    unicode[3596]:=16#75c8;
    unicode[3597]:=16#75c9;
    unicode[3598]:=16#75ca;
    unicode[3599]:=16#75cd;
    unicode[3600]:=16#75d2;
    unicode[3601]:=16#75d4;
    unicode[3602]:=16#75d5;
    unicode[3603]:=16#75d6;
    unicode[3604]:=16#75d8;
    unicode[3605]:=16#75db;
    unicode[3606]:=16#75de;
    unicode[3607]:=16#75e2;
    unicode[3608]:=16#75e3;
    unicode[3609]:=16#75e4;
    unicode[3610]:=16#75e6;
    unicode[3611]:=16#75e7;
    unicode[3612]:=16#75e8;
    unicode[3613]:=16#75ea;
    unicode[3614]:=16#75eb;
    unicode[3615]:=16#75f0;
    unicode[3616]:=16#75f1;
    unicode[3617]:=16#75f4;
    unicode[3618]:=16#75f9;
    unicode[3619]:=16#75fc;
    unicode[3620]:=16#75ff;
    unicode[3621]:=16#7600;
    unicode[3622]:=16#7601;
    unicode[3623]:=16#7603;
    unicode[3624]:=16#7605;
    unicode[3625]:=16#760a;
    unicode[3626]:=16#760c;
    unicode[3627]:=16#7610;
    unicode[3628]:=16#7615;
    unicode[3629]:=16#7617;
    unicode[3630]:=16#7618;
    unicode[3631]:=16#7619;
    unicode[3632]:=16#761b;
    unicode[3633]:=16#761f;
    unicode[3634]:=16#7620;
    unicode[3635]:=16#7622;
    unicode[3636]:=16#7624;
    unicode[3637]:=16#7625;
    unicode[3638]:=16#7626;
    unicode[3639]:=16#7629;
    unicode[3640]:=16#762a;
    unicode[3641]:=16#762b;
    unicode[3642]:=16#762d;
    unicode[3643]:=16#7630;
    unicode[3644]:=16#7633;
    unicode[3645]:=16#7634;
    unicode[3646]:=16#7635;
    unicode[3647]:=16#7638;
    unicode[3648]:=16#763c;
    unicode[3649]:=16#763e;
    unicode[3650]:=16#763f;
    unicode[3651]:=16#7640;
    unicode[3652]:=16#7643;
    unicode[3653]:=16#764c;
    unicode[3654]:=16#764d;
    unicode[3655]:=16#7654;
    unicode[3656]:=16#7656;
    unicode[3657]:=16#765c;
    unicode[3658]:=16#765e;
    unicode[3659]:=16#7663;
    unicode[3660]:=16#766b;
    unicode[3661]:=16#766f;
    unicode[3662]:=16#7678;
    unicode[3663]:=16#767b;
    unicode[3664]:=16#767d;
    unicode[3665]:=16#767e;
    unicode[3666]:=16#7682;
    unicode[3667]:=16#7684;
    unicode[3668]:=16#7686;
    unicode[3669]:=16#7687;
    unicode[3670]:=16#7688;
    unicode[3671]:=16#768b;
    unicode[3672]:=16#768e;
    unicode[3673]:=16#7691;
    unicode[3674]:=16#7693;
    unicode[3675]:=16#7696;
    unicode[3676]:=16#7699;
    unicode[3677]:=16#76a4;
    unicode[3678]:=16#76ae;
    unicode[3679]:=16#76b1;
    unicode[3680]:=16#76b2;
    unicode[3681]:=16#76b4;
    unicode[3682]:=16#76bf;
    unicode[3683]:=16#76c2;
    unicode[3684]:=16#76c5;
    unicode[3685]:=16#76c6;
    unicode[3686]:=16#76c8;
    unicode[3687]:=16#76ca;
    unicode[3688]:=16#76cd;
    unicode[3689]:=16#76ce;
    unicode[3690]:=16#76cf;
    unicode[3691]:=16#76d0;
    unicode[3692]:=16#76d1;
    unicode[3693]:=16#76d2;
    unicode[3694]:=16#76d4;
    unicode[3695]:=16#76d6;
    unicode[3696]:=16#76d7;
    unicode[3697]:=16#76d8;
    unicode[3698]:=16#76db;
    unicode[3699]:=16#76df;
    unicode[3700]:=16#76e5;
    unicode[3701]:=16#76ee;
    unicode[3702]:=16#76ef;
    unicode[3703]:=16#76f1;
    unicode[3704]:=16#76f2;
    unicode[3705]:=16#76f4;
    unicode[3706]:=16#76f8;
    unicode[3707]:=16#76f9;
    unicode[3708]:=16#76fc;
    unicode[3709]:=16#76fe;
    unicode[3710]:=16#7701;
    unicode[3711]:=16#7704;
    unicode[3712]:=16#7707;
    unicode[3713]:=16#7708;
    unicode[3714]:=16#7709;
    unicode[3715]:=16#770b;
    unicode[3716]:=16#770d;
    unicode[3717]:=16#7719;
    unicode[3718]:=16#771a;
    unicode[3719]:=16#771f;
    unicode[3720]:=16#7720;
    unicode[3721]:=16#7722;
    unicode[3722]:=16#7726;
    unicode[3723]:=16#7728;
    unicode[3724]:=16#7729;
    unicode[3725]:=16#772d;
    unicode[3726]:=16#772f;
    unicode[3727]:=16#7735;
    unicode[3728]:=16#7736;
    unicode[3729]:=16#7737;
    unicode[3730]:=16#7738;
    unicode[3731]:=16#773a;
    unicode[3732]:=16#773c;
    unicode[3733]:=16#7740;
    unicode[3734]:=16#7741;
    unicode[3735]:=16#7743;
    unicode[3736]:=16#7747;
    unicode[3737]:=16#7750;
    unicode[3738]:=16#7751;
    unicode[3739]:=16#775a;
    unicode[3740]:=16#775b;
    unicode[3741]:=16#7761;
    unicode[3742]:=16#7762;
    unicode[3743]:=16#7763;
    unicode[3744]:=16#7765;
    unicode[3745]:=16#7766;
    unicode[3746]:=16#7768;
    unicode[3747]:=16#776b;
    unicode[3748]:=16#776c;
    unicode[3749]:=16#7779;
    unicode[3750]:=16#777d;
    unicode[3751]:=16#777e;
    unicode[3752]:=16#777f;
    unicode[3753]:=16#7780;
    unicode[3754]:=16#7784;
    unicode[3755]:=16#7785;
    unicode[3756]:=16#778c;
    unicode[3757]:=16#778d;
    unicode[3758]:=16#778e;
    unicode[3759]:=16#7791;
    unicode[3760]:=16#7792;
    unicode[3761]:=16#779f;
    unicode[3762]:=16#77a0;
    unicode[3763]:=16#77a2;
    unicode[3764]:=16#77a5;
    unicode[3765]:=16#77a7;
    unicode[3766]:=16#77a9;
    unicode[3767]:=16#77aa;
    unicode[3768]:=16#77ac;
    unicode[3769]:=16#77b0;
    unicode[3770]:=16#77b3;
    unicode[3771]:=16#77b5;
    unicode[3772]:=16#77bb;
    unicode[3773]:=16#77bd;
    unicode[3774]:=16#77bf;
    unicode[3775]:=16#77cd;
    unicode[3776]:=16#77d7;
    unicode[3777]:=16#77db;
    unicode[3778]:=16#77dc;
    unicode[3779]:=16#77e2;
    unicode[3780]:=16#77e3;
    unicode[3781]:=16#77e5;
    unicode[3782]:=16#77e7;
    unicode[3783]:=16#77e9;
    unicode[3784]:=16#77eb;
    unicode[3785]:=16#77ec;
    unicode[3786]:=16#77ed;
    unicode[3787]:=16#77ee;
    unicode[3788]:=16#77f3;
    unicode[3789]:=16#77f6;
    unicode[3790]:=16#77f8;
    unicode[3791]:=16#77fd;
    unicode[3792]:=16#77fe;
    unicode[3793]:=16#77ff;
    unicode[3794]:=16#7800;
    unicode[3795]:=16#7801;
    unicode[3796]:=16#7802;
    unicode[3797]:=16#7809;
    unicode[3798]:=16#780c;
    unicode[3799]:=16#780d;
    unicode[3800]:=16#7811;
    unicode[3801]:=16#7812;
    unicode[3802]:=16#7814;
    unicode[3803]:=16#7816;
    unicode[3804]:=16#7817;
    unicode[3805]:=16#7818;
    unicode[3806]:=16#781a;
    unicode[3807]:=16#781c;
    unicode[3808]:=16#781d;
    unicode[3809]:=16#781f;
    unicode[3810]:=16#7823;
    unicode[3811]:=16#7825;
    unicode[3812]:=16#7826;
    unicode[3813]:=16#7827;
    unicode[3814]:=16#7829;
    unicode[3815]:=16#782c;
    unicode[3816]:=16#782d;
    unicode[3817]:=16#7830;
    unicode[3818]:=16#7834;
    unicode[3819]:=16#7837;
    unicode[3820]:=16#7838;
    unicode[3821]:=16#7839;
    unicode[3822]:=16#783a;
    unicode[3823]:=16#783b;
    unicode[3824]:=16#783c;
    unicode[3825]:=16#783e;
    unicode[3826]:=16#7840;
    unicode[3827]:=16#7845;
    unicode[3828]:=16#7847;
    unicode[3829]:=16#784c;
    unicode[3830]:=16#784e;
    unicode[3831]:=16#7850;
    unicode[3832]:=16#7852;
    unicode[3833]:=16#7855;
    unicode[3834]:=16#7856;
    unicode[3835]:=16#7857;
    unicode[3836]:=16#785d;
    unicode[3837]:=16#786a;
    unicode[3838]:=16#786b;
    unicode[3839]:=16#786c;
    unicode[3840]:=16#786d;
    unicode[3841]:=16#786e;
    unicode[3842]:=16#7877;
    unicode[3843]:=16#787c;
    unicode[3844]:=16#7887;
    unicode[3845]:=16#7889;
    unicode[3846]:=16#788c;
    unicode[3847]:=16#788d;
    unicode[3848]:=16#788e;
    unicode[3849]:=16#7891;
    unicode[3850]:=16#7893;
    unicode[3851]:=16#7897;
    unicode[3852]:=16#7898;
    unicode[3853]:=16#789a;
    unicode[3854]:=16#789b;
    unicode[3855]:=16#789c;
    unicode[3856]:=16#789f;
    unicode[3857]:=16#78a1;
    unicode[3858]:=16#78a3;
    unicode[3859]:=16#78a5;
    unicode[3860]:=16#78a7;
    unicode[3861]:=16#78b0;
    unicode[3862]:=16#78b1;
    unicode[3863]:=16#78b2;
    unicode[3864]:=16#78b3;
    unicode[3865]:=16#78b4;
    unicode[3866]:=16#78b9;
    unicode[3867]:=16#78be;
    unicode[3868]:=16#78c1;
    unicode[3869]:=16#78c5;
    unicode[3870]:=16#78c9;
    unicode[3871]:=16#78ca;
    unicode[3872]:=16#78cb;
    unicode[3873]:=16#78d0;
    unicode[3874]:=16#78d4;
    unicode[3875]:=16#78d5;
    unicode[3876]:=16#78d9;
    unicode[3877]:=16#78e8;
    unicode[3878]:=16#78ec;
    unicode[3879]:=16#78f2;
    unicode[3880]:=16#78f4;
    unicode[3881]:=16#78f7;
    unicode[3882]:=16#78fa;
    unicode[3883]:=16#7901;
    unicode[3884]:=16#7905;
    unicode[3885]:=16#7913;
    unicode[3886]:=16#791e;
    unicode[3887]:=16#7924;
    unicode[3888]:=16#7934;
    unicode[3889]:=16#793a;
    unicode[3890]:=16#793b;
    unicode[3891]:=16#793c;
    unicode[3892]:=16#793e;
    unicode[3893]:=16#7940;
    unicode[3894]:=16#7941;
    unicode[3895]:=16#7946;
    unicode[3896]:=16#7948;
    unicode[3897]:=16#7949;
    unicode[3898]:=16#7953;
    unicode[3899]:=16#7956;
    unicode[3900]:=16#7957;
    unicode[3901]:=16#795a;
    unicode[3902]:=16#795b;
    unicode[3903]:=16#795c;
    unicode[3904]:=16#795d;
    unicode[3905]:=16#795e;
    unicode[3906]:=16#795f;
    unicode[3907]:=16#7960;
    unicode[3908]:=16#7962;
    unicode[3909]:=16#7965;
    unicode[3910]:=16#7967;
    unicode[3911]:=16#7968;
    unicode[3912]:=16#796d;
    unicode[3913]:=16#796f;
    unicode[3914]:=16#7977;
    unicode[3915]:=16#7978;
    unicode[3916]:=16#797a;
    unicode[3917]:=16#7980;
    unicode[3918]:=16#7981;
    unicode[3919]:=16#7984;
    unicode[3920]:=16#7985;
    unicode[3921]:=16#798a;
    unicode[3922]:=16#798f;
    unicode[3923]:=16#799a;
    unicode[3924]:=16#79a7;
    unicode[3925]:=16#79b3;
    unicode[3926]:=16#79b9;
    unicode[3927]:=16#79ba;
    unicode[3928]:=16#79bb;
    unicode[3929]:=16#79bd;
    unicode[3930]:=16#79be;
    unicode[3931]:=16#79c0;
    unicode[3932]:=16#79c1;
    unicode[3933]:=16#79c3;
    unicode[3934]:=16#79c6;
    unicode[3935]:=16#79c9;
    unicode[3936]:=16#79cb;
    unicode[3937]:=16#79cd;
    unicode[3938]:=16#79d1;
    unicode[3939]:=16#79d2;
    unicode[3940]:=16#79d5;
    unicode[3941]:=16#79d8;
    unicode[3942]:=16#79df;
    unicode[3943]:=16#79e3;
    unicode[3944]:=16#79e4;
    unicode[3945]:=16#79e6;
    unicode[3946]:=16#79e7;
    unicode[3947]:=16#79e9;
    unicode[3948]:=16#79eb;
    unicode[3949]:=16#79ed;
    unicode[3950]:=16#79ef;
    unicode[3951]:=16#79f0;
    unicode[3952]:=16#79f8;
    unicode[3953]:=16#79fb;
    unicode[3954]:=16#79fd;
    unicode[3955]:=16#7a00;
    unicode[3956]:=16#7a02;
    unicode[3957]:=16#7a03;
    unicode[3958]:=16#7a06;
    unicode[3959]:=16#7a0b;
    unicode[3960]:=16#7a0d;
    unicode[3961]:=16#7a0e;
    unicode[3962]:=16#7a14;
    unicode[3963]:=16#7a17;
    unicode[3964]:=16#7a1a;
    unicode[3965]:=16#7a1e;
    unicode[3966]:=16#7a20;
    unicode[3967]:=16#7a23;
    unicode[3968]:=16#7a33;
    unicode[3969]:=16#7a37;
    unicode[3970]:=16#7a39;
    unicode[3971]:=16#7a3b;
    unicode[3972]:=16#7a3c;
    unicode[3973]:=16#7a3d;
    unicode[3974]:=16#7a3f;
    unicode[3975]:=16#7a46;
    unicode[3976]:=16#7a51;
    unicode[3977]:=16#7a57;
    unicode[3978]:=16#7a70;
    unicode[3979]:=16#7a74;
    unicode[3980]:=16#7a76;
    unicode[3981]:=16#7a77;
    unicode[3982]:=16#7a78;
    unicode[3983]:=16#7a79;
    unicode[3984]:=16#7a7a;
    unicode[3985]:=16#7a7f;
    unicode[3986]:=16#7a80;
    unicode[3987]:=16#7a81;
    unicode[3988]:=16#7a83;
    unicode[3989]:=16#7a84;
    unicode[3990]:=16#7a86;
    unicode[3991]:=16#7a88;
    unicode[3992]:=16#7a8d;
    unicode[3993]:=16#7a91;
    unicode[3994]:=16#7a92;
    unicode[3995]:=16#7a95;
    unicode[3996]:=16#7a96;
    unicode[3997]:=16#7a97;
    unicode[3998]:=16#7a98;
    unicode[3999]:=16#7a9c;               //unicode码 3000-3999
END_IF;
(* Rung 8 *)
IF P_On THEN
    unicode[4000]:=16#7a9d;
    unicode[4001]:=16#7a9f;
    unicode[4002]:=16#7aa0;
    unicode[4003]:=16#7aa5;
    unicode[4004]:=16#7aa6;
    unicode[4005]:=16#7aa8;
    unicode[4006]:=16#7aac;
    unicode[4007]:=16#7aad;
    unicode[4008]:=16#7ab3;
    unicode[4009]:=16#7abf;
    unicode[4010]:=16#7acb;
    unicode[4011]:=16#7ad6;
    unicode[4012]:=16#7ad9;
    unicode[4013]:=16#7ade;
    unicode[4014]:=16#7adf;
    unicode[4015]:=16#7ae0;
    unicode[4016]:=16#7ae3;
    unicode[4017]:=16#7ae5;
    unicode[4018]:=16#7ae6;
    unicode[4019]:=16#7aed;
    unicode[4020]:=16#7aef;
    unicode[4021]:=16#7af9;
    unicode[4022]:=16#7afa;
    unicode[4023]:=16#7afd;
    unicode[4024]:=16#7aff;
    unicode[4025]:=16#7b03;
    unicode[4026]:=16#7b04;
    unicode[4027]:=16#7b06;
    unicode[4028]:=16#7b08;
    unicode[4029]:=16#7b0a;
    unicode[4030]:=16#7b0b;
    unicode[4031]:=16#7b0f;
    unicode[4032]:=16#7b11;
    unicode[4033]:=16#7b14;
    unicode[4034]:=16#7b15;
    unicode[4035]:=16#7b19;
    unicode[4036]:=16#7b1b;
    unicode[4037]:=16#7b1e;
    unicode[4038]:=16#7b20;
    unicode[4039]:=16#7b24;
    unicode[4040]:=16#7b25;
    unicode[4041]:=16#7b26;
    unicode[4042]:=16#7b28;
    unicode[4043]:=16#7b2a;
    unicode[4044]:=16#7b2b;
    unicode[4045]:=16#7b2c;
    unicode[4046]:=16#7b2e;
    unicode[4047]:=16#7b31;
    unicode[4048]:=16#7b33;
    unicode[4049]:=16#7b38;
    unicode[4050]:=16#7b3a;
    unicode[4051]:=16#7b3c;
    unicode[4052]:=16#7b3e;
    unicode[4053]:=16#7b45;
    unicode[4054]:=16#7b47;
    unicode[4055]:=16#7b49;
    unicode[4056]:=16#7b4b;
    unicode[4057]:=16#7b4c;
    unicode[4058]:=16#7b4f;
    unicode[4059]:=16#7b50;
    unicode[4060]:=16#7b51;
    unicode[4061]:=16#7b52;
    unicode[4062]:=16#7b54;
    unicode[4063]:=16#7b56;
    unicode[4064]:=16#7b58;
    unicode[4065]:=16#7b5a;
    unicode[4066]:=16#7b5b;
    unicode[4067]:=16#7b5d;
    unicode[4068]:=16#7b60;
    unicode[4069]:=16#7b62;
    unicode[4070]:=16#7b6e;
    unicode[4071]:=16#7b71;
    unicode[4072]:=16#7b72;
    unicode[4073]:=16#7b75;
    unicode[4074]:=16#7b77;
    unicode[4075]:=16#7b79;
    unicode[4076]:=16#7b7b;
    unicode[4077]:=16#7b7e;
    unicode[4078]:=16#7b80;
    unicode[4079]:=16#7b85;
    unicode[4080]:=16#7b8d;
    unicode[4081]:=16#7b90;
    unicode[4082]:=16#7b94;
    unicode[4083]:=16#7b95;
    unicode[4084]:=16#7b97;
    unicode[4085]:=16#7b9c;
    unicode[4086]:=16#7b9d;
    unicode[4087]:=16#7ba1;
    unicode[4088]:=16#7ba2;
    unicode[4089]:=16#7ba6;
    unicode[4090]:=16#7ba7;
    unicode[4091]:=16#7ba8;
    unicode[4092]:=16#7ba9;
    unicode[4093]:=16#7baa;
    unicode[4094]:=16#7bab;
    unicode[4095]:=16#7bac;
    unicode[4096]:=16#7bad;
    unicode[4097]:=16#7bb1;
    unicode[4098]:=16#7bb4;
    unicode[4099]:=16#7bb8;
    unicode[4100]:=16#7bc1;
    unicode[4101]:=16#7bc6;
    unicode[4102]:=16#7bc7;
    unicode[4103]:=16#7bcc;
    unicode[4104]:=16#7bd1;
    unicode[4105]:=16#7bd3;
    unicode[4106]:=16#7bd9;
    unicode[4107]:=16#7bda;
    unicode[4108]:=16#7bdd;
    unicode[4109]:=16#7be1;
    unicode[4110]:=16#7be5;
    unicode[4111]:=16#7be6;
    unicode[4112]:=16#7bea;
    unicode[4113]:=16#7bee;
    unicode[4114]:=16#7bf1;
    unicode[4115]:=16#7bf7;
    unicode[4116]:=16#7bfc;
    unicode[4117]:=16#7bfe;
    unicode[4118]:=16#7c07;
    unicode[4119]:=16#7c0b;
    unicode[4120]:=16#7c0c;
    unicode[4121]:=16#7c0f;
    unicode[4122]:=16#7c16;
    unicode[4123]:=16#7c1f;
    unicode[4124]:=16#7c26;
    unicode[4125]:=16#7c27;
    unicode[4126]:=16#7c2a;
    unicode[4127]:=16#7c38;
    unicode[4128]:=16#7c3f;
    unicode[4129]:=16#7c40;
    unicode[4130]:=16#7c41;
    unicode[4131]:=16#7c4d;
    unicode[4132]:=16#7c73;
    unicode[4133]:=16#7c74;
    unicode[4134]:=16#7c7b;
    unicode[4135]:=16#7c7c;
    unicode[4136]:=16#7c7d;
    unicode[4137]:=16#7c89;
    unicode[4138]:=16#7c91;
    unicode[4139]:=16#7c92;
    unicode[4140]:=16#7c95;
    unicode[4141]:=16#7c97;
    unicode[4142]:=16#7c98;
    unicode[4143]:=16#7c9c;
    unicode[4144]:=16#7c9d;
    unicode[4145]:=16#7c9e;
    unicode[4146]:=16#7c9f;
    unicode[4147]:=16#7ca2;
    unicode[4148]:=16#7ca4;
    unicode[4149]:=16#7ca5;
    unicode[4150]:=16#7caa;
    unicode[4151]:=16#7cae;
    unicode[4152]:=16#7cb1;
    unicode[4153]:=16#7cb2;
    unicode[4154]:=16#7cb3;
    unicode[4155]:=16#7cb9;
    unicode[4156]:=16#7cbc;
    unicode[4157]:=16#7cbd;
    unicode[4158]:=16#7cbe;
    unicode[4159]:=16#7cc1;
    unicode[4160]:=16#7cc5;
    unicode[4161]:=16#7cc7;
    unicode[4162]:=16#7cc8;
    unicode[4163]:=16#7cca;
    unicode[4164]:=16#7ccc;
    unicode[4165]:=16#7ccd;
    unicode[4166]:=16#7cd5;
    unicode[4167]:=16#7cd6;
    unicode[4168]:=16#7cd7;
    unicode[4169]:=16#7cd9;
    unicode[4170]:=16#7cdc;
    unicode[4171]:=16#7cdf;
    unicode[4172]:=16#7ce0;
    unicode[4173]:=16#7ce8;
    unicode[4174]:=16#7cef;
    unicode[4175]:=16#7cf8;
    unicode[4176]:=16#7cfb;
    unicode[4177]:=16#7d0a;
    unicode[4178]:=16#7d20;
    unicode[4179]:=16#7d22;
    unicode[4180]:=16#7d27;
    unicode[4181]:=16#7d2b;
    unicode[4182]:=16#7d2f;
    unicode[4183]:=16#7d6e;
    unicode[4184]:=16#7d77;
    unicode[4185]:=16#7da6;
    unicode[4186]:=16#7dae;
    unicode[4187]:=16#7e3b;
    unicode[4188]:=16#7e41;
    unicode[4189]:=16#7e47;
    unicode[4190]:=16#7e82;
    unicode[4191]:=16#7e9b;
    unicode[4192]:=16#7e9f;
    unicode[4193]:=16#7ea0;
    unicode[4194]:=16#7ea1;
    unicode[4195]:=16#7ea2;
    unicode[4196]:=16#7ea3;
    unicode[4197]:=16#7ea4;
    unicode[4198]:=16#7ea5;
    unicode[4199]:=16#7ea6;
    unicode[4200]:=16#7ea7;
    unicode[4201]:=16#7ea8;
    unicode[4202]:=16#7ea9;
    unicode[4203]:=16#7eaa;
    unicode[4204]:=16#7eab;
    unicode[4205]:=16#7eac;
    unicode[4206]:=16#7ead;
    unicode[4207]:=16#7eaf;
    unicode[4208]:=16#7eb0;
    unicode[4209]:=16#7eb1;
    unicode[4210]:=16#7eb2;
    unicode[4211]:=16#7eb3;
    unicode[4212]:=16#7eb5;
    unicode[4213]:=16#7eb6;
    unicode[4214]:=16#7eb7;
    unicode[4215]:=16#7eb8;
    unicode[4216]:=16#7eb9;
    unicode[4217]:=16#7eba;
    unicode[4218]:=16#7ebd;
    unicode[4219]:=16#7ebe;
    unicode[4220]:=16#7ebf;
    unicode[4221]:=16#7ec0;
    unicode[4222]:=16#7ec1;
    unicode[4223]:=16#7ec2;
    unicode[4224]:=16#7ec3;
    unicode[4225]:=16#7ec4;
    unicode[4226]:=16#7ec5;
    unicode[4227]:=16#7ec6;
    unicode[4228]:=16#7ec7;
    unicode[4229]:=16#7ec8;
    unicode[4230]:=16#7ec9;
    unicode[4231]:=16#7eca;
    unicode[4232]:=16#7ecb;
    unicode[4233]:=16#7ecc;
    unicode[4234]:=16#7ecd;
    unicode[4235]:=16#7ece;
    unicode[4236]:=16#7ecf;
    unicode[4237]:=16#7ed0;
    unicode[4238]:=16#7ed1;
    unicode[4239]:=16#7ed2;
    unicode[4240]:=16#7ed3;
    unicode[4241]:=16#7ed4;
    unicode[4242]:=16#7ed5;
    unicode[4243]:=16#7ed7;
    unicode[4244]:=16#7ed8;
    unicode[4245]:=16#7ed9;
    unicode[4246]:=16#7eda;
    unicode[4247]:=16#7edb;
    unicode[4248]:=16#7edc;
    unicode[4249]:=16#7edd;
    unicode[4250]:=16#7ede;
    unicode[4251]:=16#7edf;
    unicode[4252]:=16#7ee0;
    unicode[4253]:=16#7ee1;
    unicode[4254]:=16#7ee2;
    unicode[4255]:=16#7ee3;
    unicode[4256]:=16#7ee5;
    unicode[4257]:=16#7ee6;
    unicode[4258]:=16#7ee7;
    unicode[4259]:=16#7ee8;
    unicode[4260]:=16#7ee9;
    unicode[4261]:=16#7eea;
    unicode[4262]:=16#7eeb;
    unicode[4263]:=16#7eed;
    unicode[4264]:=16#7eee;
    unicode[4265]:=16#7eef;
    unicode[4266]:=16#7ef0;
    unicode[4267]:=16#7ef1;
    unicode[4268]:=16#7ef2;
    unicode[4269]:=16#7ef3;
    unicode[4270]:=16#7ef4;
    unicode[4271]:=16#7ef5;
    unicode[4272]:=16#7ef6;
    unicode[4273]:=16#7ef7;
    unicode[4274]:=16#7ef8;
    unicode[4275]:=16#7efa;
    unicode[4276]:=16#7efb;
    unicode[4277]:=16#7efc;
    unicode[4278]:=16#7efd;
    unicode[4279]:=16#7efe;
    unicode[4280]:=16#7eff;
    unicode[4281]:=16#7f00;
    unicode[4282]:=16#7f01;
    unicode[4283]:=16#7f02;
    unicode[4284]:=16#7f03;
    unicode[4285]:=16#7f04;
    unicode[4286]:=16#7f05;
    unicode[4287]:=16#7f06;
    unicode[4288]:=16#7f07;
    unicode[4289]:=16#7f08;
    unicode[4290]:=16#7f09;
    unicode[4291]:=16#7f0b;
    unicode[4292]:=16#7f0c;
    unicode[4293]:=16#7f0d;
    unicode[4294]:=16#7f0e;
    unicode[4295]:=16#7f0f;
    unicode[4296]:=16#7f11;
    unicode[4297]:=16#7f12;
    unicode[4298]:=16#7f13;
    unicode[4299]:=16#7f14;
    unicode[4300]:=16#7f15;
    unicode[4301]:=16#7f16;
    unicode[4302]:=16#7f17;
    unicode[4303]:=16#7f18;
    unicode[4304]:=16#7f19;
    unicode[4305]:=16#7f1a;
    unicode[4306]:=16#7f1b;
    unicode[4307]:=16#7f1c;
    unicode[4308]:=16#7f1d;
    unicode[4309]:=16#7f1f;
    unicode[4310]:=16#7f20;
    unicode[4311]:=16#7f21;
    unicode[4312]:=16#7f22;
    unicode[4313]:=16#7f23;
    unicode[4314]:=16#7f24;
    unicode[4315]:=16#7f25;
    unicode[4316]:=16#7f26;
    unicode[4317]:=16#7f27;
    unicode[4318]:=16#7f28;
    unicode[4319]:=16#7f29;
    unicode[4320]:=16#7f2a;
    unicode[4321]:=16#7f2b;
    unicode[4322]:=16#7f2c;
    unicode[4323]:=16#7f2d;
    unicode[4324]:=16#7f2e;
    unicode[4325]:=16#7f2f;
    unicode[4326]:=16#7f30;
    unicode[4327]:=16#7f31;
    unicode[4328]:=16#7f32;
    unicode[4329]:=16#7f33;
    unicode[4330]:=16#7f34;
    unicode[4331]:=16#7f35;
    unicode[4332]:=16#7f36;
    unicode[4333]:=16#7f38;
    unicode[4334]:=16#7f3a;
    unicode[4335]:=16#7f42;
    unicode[4336]:=16#7f44;
    unicode[4337]:=16#7f45;
    unicode[4338]:=16#7f50;
    unicode[4339]:=16#7f51;
    unicode[4340]:=16#7f54;
    unicode[4341]:=16#7f55;
    unicode[4342]:=16#7f57;
    unicode[4343]:=16#7f58;
    unicode[4344]:=16#7f5a;
    unicode[4345]:=16#7f5f;
    unicode[4346]:=16#7f61;
    unicode[4347]:=16#7f62;
    unicode[4348]:=16#7f68;
    unicode[4349]:=16#7f69;
    unicode[4350]:=16#7f6a;
    unicode[4351]:=16#7f6e;
    unicode[4352]:=16#7f71;
    unicode[4353]:=16#7f72;
    unicode[4354]:=16#7f74;
    unicode[4355]:=16#7f79;
    unicode[4356]:=16#7f7e;
    unicode[4357]:=16#7f81;
    unicode[4358]:=16#7f8a;
    unicode[4359]:=16#7f8c;
    unicode[4360]:=16#7f8e;
    unicode[4361]:=16#7f94;
    unicode[4362]:=16#7f9a;
    unicode[4363]:=16#7f9d;
    unicode[4364]:=16#7f9e;
    unicode[4365]:=16#7f9f;
    unicode[4366]:=16#7fa1;
    unicode[4367]:=16#7fa4;
    unicode[4368]:=16#7fa7;
    unicode[4369]:=16#7faf;
    unicode[4370]:=16#7fb0;
    unicode[4371]:=16#7fb2;
    unicode[4372]:=16#7fb8;
    unicode[4373]:=16#7fb9;
    unicode[4374]:=16#7fbc;
    unicode[4375]:=16#7fbd;
    unicode[4376]:=16#7fbf;
    unicode[4377]:=16#7fc1;
    unicode[4378]:=16#7fc5;
    unicode[4379]:=16#7fca;
    unicode[4380]:=16#7fcc;
    unicode[4381]:=16#7fce;
    unicode[4382]:=16#7fd4;
    unicode[4383]:=16#7fd5;
    unicode[4384]:=16#7fd8;
    unicode[4385]:=16#7fdf;
    unicode[4386]:=16#7fe0;
    unicode[4387]:=16#7fe1;
    unicode[4388]:=16#7fe5;
    unicode[4389]:=16#7fe6;
    unicode[4390]:=16#7fe9;
    unicode[4391]:=16#7fee;
    unicode[4392]:=16#7ff0;
    unicode[4393]:=16#7ff1;
    unicode[4394]:=16#7ff3;
    unicode[4395]:=16#7ffb;
    unicode[4396]:=16#7ffc;
    unicode[4397]:=16#8000;
    unicode[4398]:=16#8001;
    unicode[4399]:=16#8003;
    unicode[4400]:=16#8004;
    unicode[4401]:=16#8005;
    unicode[4402]:=16#8006;
    unicode[4403]:=16#800b;
    unicode[4404]:=16#800c;
    unicode[4405]:=16#800d;
    unicode[4406]:=16#8010;
    unicode[4407]:=16#8012;
    unicode[4408]:=16#8014;
    unicode[4409]:=16#8015;
    unicode[4410]:=16#8016;
    unicode[4411]:=16#8017;
    unicode[4412]:=16#8018;
    unicode[4413]:=16#8019;
    unicode[4414]:=16#801c;
    unicode[4415]:=16#8020;
    unicode[4416]:=16#8022;
    unicode[4417]:=16#8025;
    unicode[4418]:=16#8026;
    unicode[4419]:=16#8027;
    unicode[4420]:=16#8028;
    unicode[4421]:=16#8029;
    unicode[4422]:=16#802a;
    unicode[4423]:=16#8031;
    unicode[4424]:=16#8033;
    unicode[4425]:=16#8035;
    unicode[4426]:=16#8036;
    unicode[4427]:=16#8037;
    unicode[4428]:=16#8038;
    unicode[4429]:=16#803b;
    unicode[4430]:=16#803d;
    unicode[4431]:=16#803f;
    unicode[4432]:=16#8042;
    unicode[4433]:=16#8043;
    unicode[4434]:=16#8046;
    unicode[4435]:=16#804a;
    unicode[4436]:=16#804b;
    unicode[4437]:=16#804c;
    unicode[4438]:=16#804d;
    unicode[4439]:=16#8052;
    unicode[4440]:=16#8054;
    unicode[4441]:=16#8058;
    unicode[4442]:=16#805a;
    unicode[4443]:=16#8069;
    unicode[4444]:=16#806a;
    unicode[4445]:=16#8071;
    unicode[4446]:=16#807f;
    unicode[4447]:=16#8080;
    unicode[4448]:=16#8083;
    unicode[4449]:=16#8084;
    unicode[4450]:=16#8086;
    unicode[4451]:=16#8087;
    unicode[4452]:=16#8089;
    unicode[4453]:=16#808b;
    unicode[4454]:=16#808c;
    unicode[4455]:=16#8093;
    unicode[4456]:=16#8096;
    unicode[4457]:=16#8098;
    unicode[4458]:=16#809a;
    unicode[4459]:=16#809b;
    unicode[4460]:=16#809c;
    unicode[4461]:=16#809d;
    unicode[4462]:=16#809f;
    unicode[4463]:=16#80a0;
    unicode[4464]:=16#80a1;
    unicode[4465]:=16#80a2;
    unicode[4466]:=16#80a4;
    unicode[4467]:=16#80a5;
    unicode[4468]:=16#80a9;
    unicode[4469]:=16#80aa;
    unicode[4470]:=16#80ab;
    unicode[4471]:=16#80ad;
    unicode[4472]:=16#80ae;
    unicode[4473]:=16#80af;
    unicode[4474]:=16#80b1;
    unicode[4475]:=16#80b2;
    unicode[4476]:=16#80b4;
    unicode[4477]:=16#80b7;
    unicode[4478]:=16#80ba;
    unicode[4479]:=16#80bc;
    unicode[4480]:=16#80bd;
    unicode[4481]:=16#80be;
    unicode[4482]:=16#80bf;
    unicode[4483]:=16#80c0;
    unicode[4484]:=16#80c1;
    unicode[4485]:=16#80c2;
    unicode[4486]:=16#80c3;
    unicode[4487]:=16#80c4;
    unicode[4488]:=16#80c6;
    unicode[4489]:=16#80cc;
    unicode[4490]:=16#80cd;
    unicode[4491]:=16#80ce;
    unicode[4492]:=16#80d6;
    unicode[4493]:=16#80d7;
    unicode[4494]:=16#80d9;
    unicode[4495]:=16#80da;
    unicode[4496]:=16#80db;
    unicode[4497]:=16#80dc;
    unicode[4498]:=16#80dd;
    unicode[4499]:=16#80de;
    unicode[4500]:=16#80e1;
    unicode[4501]:=16#80e4;
    unicode[4502]:=16#80e5;
    unicode[4503]:=16#80e7;
    unicode[4504]:=16#80e8;
    unicode[4505]:=16#80e9;
    unicode[4506]:=16#80ea;
    unicode[4507]:=16#80eb;
    unicode[4508]:=16#80ec;
    unicode[4509]:=16#80ed;
    unicode[4510]:=16#80ef;
    unicode[4511]:=16#80f0;
    unicode[4512]:=16#80f1;
    unicode[4513]:=16#80f2;
    unicode[4514]:=16#80f3;
    unicode[4515]:=16#80f4;
    unicode[4516]:=16#80f6;
    unicode[4517]:=16#80f8;
    unicode[4518]:=16#80fa;
    unicode[4519]:=16#80fc;
    unicode[4520]:=16#80fd;
    unicode[4521]:=16#8102;
    unicode[4522]:=16#8106;
    unicode[4523]:=16#8109;
    unicode[4524]:=16#810a;
    unicode[4525]:=16#810d;
    unicode[4526]:=16#810e;
    unicode[4527]:=16#810f;
    unicode[4528]:=16#8110;
    unicode[4529]:=16#8111;
    unicode[4530]:=16#8112;
    unicode[4531]:=16#8113;
    unicode[4532]:=16#8114;
    unicode[4533]:=16#8116;
    unicode[4534]:=16#8118;
    unicode[4535]:=16#811a;
    unicode[4536]:=16#811e;
    unicode[4537]:=16#812c;
    unicode[4538]:=16#812f;
    unicode[4539]:=16#8131;
    unicode[4540]:=16#8132;
    unicode[4541]:=16#8136;
    unicode[4542]:=16#8138;
    unicode[4543]:=16#813e;
    unicode[4544]:=16#8146;
    unicode[4545]:=16#8148;
    unicode[4546]:=16#814a;
    unicode[4547]:=16#814b;
    unicode[4548]:=16#814c;
    unicode[4549]:=16#8150;
    unicode[4550]:=16#8151;
    unicode[4551]:=16#8153;
    unicode[4552]:=16#8154;
    unicode[4553]:=16#8155;
    unicode[4554]:=16#8159;
    unicode[4555]:=16#815a;
    unicode[4556]:=16#8160;
    unicode[4557]:=16#8165;
    unicode[4558]:=16#8167;
    unicode[4559]:=16#8169;
    unicode[4560]:=16#816d;
    unicode[4561]:=16#816e;
    unicode[4562]:=16#8170;
    unicode[4563]:=16#8171;
    unicode[4564]:=16#8174;
    unicode[4565]:=16#8179;
    unicode[4566]:=16#817a;
    unicode[4567]:=16#817b;
    unicode[4568]:=16#817c;
    unicode[4569]:=16#817d;
    unicode[4570]:=16#817e;
    unicode[4571]:=16#817f;
    unicode[4572]:=16#8180;
    unicode[4573]:=16#8182;
    unicode[4574]:=16#8188;
    unicode[4575]:=16#818a;
    unicode[4576]:=16#818f;
    unicode[4577]:=16#8191;
    unicode[4578]:=16#8198;
    unicode[4579]:=16#819b;
    unicode[4580]:=16#819c;
    unicode[4581]:=16#819d;
    unicode[4582]:=16#81a3;
    unicode[4583]:=16#81a6;
    unicode[4584]:=16#81a8;
    unicode[4585]:=16#81aa;
    unicode[4586]:=16#81b3;
    unicode[4587]:=16#81ba;
    unicode[4588]:=16#81bb;
    unicode[4589]:=16#81c0;
    unicode[4590]:=16#81c1;
    unicode[4591]:=16#81c2;
    unicode[4592]:=16#81c3;
    unicode[4593]:=16#81c6;
    unicode[4594]:=16#81ca;
    unicode[4595]:=16#81cc;
    unicode[4596]:=16#81e3;
    unicode[4597]:=16#81e7;
    unicode[4598]:=16#81ea;
    unicode[4599]:=16#81ec;
    unicode[4600]:=16#81ed;
    unicode[4601]:=16#81f3;
    unicode[4602]:=16#81f4;
    unicode[4603]:=16#81fb;
    unicode[4604]:=16#81fc;
    unicode[4605]:=16#81fe;
    unicode[4606]:=16#8200;
    unicode[4607]:=16#8201;
    unicode[4608]:=16#8202;
    unicode[4609]:=16#8204;
    unicode[4610]:=16#8205;
    unicode[4611]:=16#8206;
    unicode[4612]:=16#820c;
    unicode[4613]:=16#820d;
    unicode[4614]:=16#8210;
    unicode[4615]:=16#8212;
    unicode[4616]:=16#8214;
    unicode[4617]:=16#821b;
    unicode[4618]:=16#821c;
    unicode[4619]:=16#821e;
    unicode[4620]:=16#821f;
    unicode[4621]:=16#8221;
    unicode[4622]:=16#8222;
    unicode[4623]:=16#8223;
    unicode[4624]:=16#8228;
    unicode[4625]:=16#822a;
    unicode[4626]:=16#822b;
    unicode[4627]:=16#822c;
    unicode[4628]:=16#822d;
    unicode[4629]:=16#822f;
    unicode[4630]:=16#8230;
    unicode[4631]:=16#8231;
    unicode[4632]:=16#8233;
    unicode[4633]:=16#8234;
    unicode[4634]:=16#8235;
    unicode[4635]:=16#8236;
    unicode[4636]:=16#8237;
    unicode[4637]:=16#8238;
    unicode[4638]:=16#8239;
    unicode[4639]:=16#823b;
    unicode[4640]:=16#823e;
    unicode[4641]:=16#8244;
    unicode[4642]:=16#8247;
    unicode[4643]:=16#8249;
    unicode[4644]:=16#824b;
    unicode[4645]:=16#824f;
    unicode[4646]:=16#8258;
    unicode[4647]:=16#825a;
    unicode[4648]:=16#825f;
    unicode[4649]:=16#8268;
    unicode[4650]:=16#826e;
    unicode[4651]:=16#826f;
    unicode[4652]:=16#8270;
    unicode[4653]:=16#8272;
    unicode[4654]:=16#8273;
    unicode[4655]:=16#8274;
    unicode[4656]:=16#8279;
    unicode[4657]:=16#827a;
    unicode[4658]:=16#827d;
    unicode[4659]:=16#827e;
    unicode[4660]:=16#827f;
    unicode[4661]:=16#8282;
    unicode[4662]:=16#8284;
    unicode[4663]:=16#8288;
    unicode[4664]:=16#828a;
    unicode[4665]:=16#828b;
    unicode[4666]:=16#828d;
    unicode[4667]:=16#828e;
    unicode[4668]:=16#828f;
    unicode[4669]:=16#8291;
    unicode[4670]:=16#8292;
    unicode[4671]:=16#8297;
    unicode[4672]:=16#8298;
    unicode[4673]:=16#8299;
    unicode[4674]:=16#829c;
    unicode[4675]:=16#829d;
    unicode[4676]:=16#829f;
    unicode[4677]:=16#82a1;
    unicode[4678]:=16#82a4;
    unicode[4679]:=16#82a5;
    unicode[4680]:=16#82a6;
    unicode[4681]:=16#82a8;
    unicode[4682]:=16#82a9;
    unicode[4683]:=16#82aa;
    unicode[4684]:=16#82ab;
    unicode[4685]:=16#82ac;
    unicode[4686]:=16#82ad;
    unicode[4687]:=16#82ae;
    unicode[4688]:=16#82af;
    unicode[4689]:=16#82b0;
    unicode[4690]:=16#82b1;
    unicode[4691]:=16#82b3;
    unicode[4692]:=16#82b4;
    unicode[4693]:=16#82b7;
    unicode[4694]:=16#82b8;
    unicode[4695]:=16#82b9;
    unicode[4696]:=16#82bd;
    unicode[4697]:=16#82be;
    unicode[4698]:=16#82c1;
    unicode[4699]:=16#82c4;
    unicode[4700]:=16#82c7;
    unicode[4701]:=16#82c8;
    unicode[4702]:=16#82ca;
    unicode[4703]:=16#82cb;
    unicode[4704]:=16#82cc;
    unicode[4705]:=16#82cd;
    unicode[4706]:=16#82ce;
    unicode[4707]:=16#82cf;
    unicode[4708]:=16#82d1;
    unicode[4709]:=16#82d2;
    unicode[4710]:=16#82d3;
    unicode[4711]:=16#82d4;
    unicode[4712]:=16#82d5;
    unicode[4713]:=16#82d7;
    unicode[4714]:=16#82d8;
    unicode[4715]:=16#82db;
    unicode[4716]:=16#82dc;
    unicode[4717]:=16#82de;
    unicode[4718]:=16#82df;
    unicode[4719]:=16#82e0;
    unicode[4720]:=16#82e1;
    unicode[4721]:=16#82e3;
    unicode[4722]:=16#82e4;
    unicode[4723]:=16#82e5;
    unicode[4724]:=16#82e6;
    unicode[4725]:=16#82eb;
    unicode[4726]:=16#82ef;
    unicode[4727]:=16#82f1;
    unicode[4728]:=16#82f4;
    unicode[4729]:=16#82f7;
    unicode[4730]:=16#82f9;
    unicode[4731]:=16#82fb;
    unicode[4732]:=16#8301;
    unicode[4733]:=16#8302;
    unicode[4734]:=16#8303;
    unicode[4735]:=16#8304;
    unicode[4736]:=16#8305;
    unicode[4737]:=16#8306;
    unicode[4738]:=16#8307;
    unicode[4739]:=16#8308;
    unicode[4740]:=16#8309;
    unicode[4741]:=16#830c;
    unicode[4742]:=16#830e;
    unicode[4743]:=16#830f;
    unicode[4744]:=16#8311;
    unicode[4745]:=16#8314;
    unicode[4746]:=16#8315;
    unicode[4747]:=16#8317;
    unicode[4748]:=16#831a;
    unicode[4749]:=16#831b;
    unicode[4750]:=16#831c;
    unicode[4751]:=16#8327;
    unicode[4752]:=16#8328;
    unicode[4753]:=16#832b;
    unicode[4754]:=16#832c;
    unicode[4755]:=16#832d;
    unicode[4756]:=16#832f;
    unicode[4757]:=16#8331;
    unicode[4758]:=16#8333;
    unicode[4759]:=16#8334;
    unicode[4760]:=16#8335;
    unicode[4761]:=16#8336;
    unicode[4762]:=16#8338;
    unicode[4763]:=16#8339;
    unicode[4764]:=16#833a;
    unicode[4765]:=16#833c;
    unicode[4766]:=16#8340;
    unicode[4767]:=16#8343;
    unicode[4768]:=16#8346;
    unicode[4769]:=16#8347;
    unicode[4770]:=16#8349;
    unicode[4771]:=16#834f;
    unicode[4772]:=16#8350;
    unicode[4773]:=16#8351;
    unicode[4774]:=16#8352;
    unicode[4775]:=16#8354;
    unicode[4776]:=16#835a;
    unicode[4777]:=16#835b;
    unicode[4778]:=16#835c;
    unicode[4779]:=16#835e;
    unicode[4780]:=16#835f;
    unicode[4781]:=16#8360;
    unicode[4782]:=16#8361;
    unicode[4783]:=16#8363;
    unicode[4784]:=16#8364;
    unicode[4785]:=16#8365;
    unicode[4786]:=16#8366;
    unicode[4787]:=16#8367;
    unicode[4788]:=16#8368;
    unicode[4789]:=16#8369;
    unicode[4790]:=16#836a;
    unicode[4791]:=16#836b;
    unicode[4792]:=16#836c;
    unicode[4793]:=16#836d;
    unicode[4794]:=16#836e;
    unicode[4795]:=16#836f;
    unicode[4796]:=16#8377;
    unicode[4797]:=16#8378;
    unicode[4798]:=16#837b;
    unicode[4799]:=16#837c;
    unicode[4800]:=16#837d;
    unicode[4801]:=16#8385;
    unicode[4802]:=16#8386;
    unicode[4803]:=16#8389;
    unicode[4804]:=16#838e;
    unicode[4805]:=16#8392;
    unicode[4806]:=16#8393;
    unicode[4807]:=16#8398;
    unicode[4808]:=16#839b;
    unicode[4809]:=16#839c;
    unicode[4810]:=16#839e;
    unicode[4811]:=16#83a0;
    unicode[4812]:=16#83a8;
    unicode[4813]:=16#83a9;
    unicode[4814]:=16#83aa;
    unicode[4815]:=16#83ab;
    unicode[4816]:=16#83b0;
    unicode[4817]:=16#83b1;
    unicode[4818]:=16#83b2;
    unicode[4819]:=16#83b3;
    unicode[4820]:=16#83b4;
    unicode[4821]:=16#83b6;
    unicode[4822]:=16#83b7;
    unicode[4823]:=16#83b8;
    unicode[4824]:=16#83b9;
    unicode[4825]:=16#83ba;
    unicode[4826]:=16#83bc;
    unicode[4827]:=16#83bd;
    unicode[4828]:=16#83c0;
    unicode[4829]:=16#83c1;
    unicode[4830]:=16#83c5;
    unicode[4831]:=16#83c7;
    unicode[4832]:=16#83ca;
    unicode[4833]:=16#83cc;
    unicode[4834]:=16#83cf;
    unicode[4835]:=16#83d4;
    unicode[4836]:=16#83d6;
    unicode[4837]:=16#83d8;
    unicode[4838]:=16#83dc;
    unicode[4839]:=16#83dd;
    unicode[4840]:=16#83df;
    unicode[4841]:=16#83e0;
    unicode[4842]:=16#83e1;
    unicode[4843]:=16#83e5;
    unicode[4844]:=16#83e9;
    unicode[4845]:=16#83ea;
    unicode[4846]:=16#83f0;
    unicode[4847]:=16#83f1;
    unicode[4848]:=16#83f2;
    unicode[4849]:=16#83f8;
    unicode[4850]:=16#83f9;
    unicode[4851]:=16#83fd;
    unicode[4852]:=16#8401;
    unicode[4853]:=16#8403;
    unicode[4854]:=16#8404;
    unicode[4855]:=16#8406;
    unicode[4856]:=16#840b;
    unicode[4857]:=16#840c;
    unicode[4858]:=16#840d;
    unicode[4859]:=16#840e;
    unicode[4860]:=16#840f;
    unicode[4861]:=16#8411;
    unicode[4862]:=16#8418;
    unicode[4863]:=16#841c;
    unicode[4864]:=16#841d;
    unicode[4865]:=16#8424;
    unicode[4866]:=16#8425;
    unicode[4867]:=16#8426;
    unicode[4868]:=16#8427;
    unicode[4869]:=16#8428;
    unicode[4870]:=16#8431;
    unicode[4871]:=16#8438;
    unicode[4872]:=16#843c;
    unicode[4873]:=16#843d;
    unicode[4874]:=16#8446;
    unicode[4875]:=16#8451;
    unicode[4876]:=16#8457;
    unicode[4877]:=16#8459;
    unicode[4878]:=16#845a;
    unicode[4879]:=16#845b;
    unicode[4880]:=16#845c;
    unicode[4881]:=16#8461;
    unicode[4882]:=16#8463;
    unicode[4883]:=16#8469;
    unicode[4884]:=16#846b;
    unicode[4885]:=16#846c;
    unicode[4886]:=16#846d;
    unicode[4887]:=16#8471;
    unicode[4888]:=16#8473;
    unicode[4889]:=16#8475;
    unicode[4890]:=16#8476;
    unicode[4891]:=16#8478;
    unicode[4892]:=16#847a;
    unicode[4893]:=16#8482;
    unicode[4894]:=16#8487;
    unicode[4895]:=16#8488;
    unicode[4896]:=16#8489;
    unicode[4897]:=16#848b;
    unicode[4898]:=16#848c;
    unicode[4899]:=16#848e;
    unicode[4900]:=16#8497;
    unicode[4901]:=16#8499;
    unicode[4902]:=16#849c;
    unicode[4903]:=16#84a1;
    unicode[4904]:=16#84af;
    unicode[4905]:=16#84b2;
    unicode[4906]:=16#84b4;
    unicode[4907]:=16#84b8;
    unicode[4908]:=16#84b9;
    unicode[4909]:=16#84ba;
    unicode[4910]:=16#84bd;
    unicode[4911]:=16#84bf;
    unicode[4912]:=16#84c1;
    unicode[4913]:=16#84c4;
    unicode[4914]:=16#84c9;
    unicode[4915]:=16#84ca;
    unicode[4916]:=16#84cd;
    unicode[4917]:=16#84d0;
    unicode[4918]:=16#84d1;
    unicode[4919]:=16#84d3;
    unicode[4920]:=16#84d6;
    unicode[4921]:=16#84dd;
    unicode[4922]:=16#84df;
    unicode[4923]:=16#84e0;
    unicode[4924]:=16#84e3;
    unicode[4925]:=16#84e5;
    unicode[4926]:=16#84e6;
    unicode[4927]:=16#84ec;
    unicode[4928]:=16#84f0;
    unicode[4929]:=16#84fc;
    unicode[4930]:=16#84ff;
    unicode[4931]:=16#850c;
    unicode[4932]:=16#8511;
    unicode[4933]:=16#8513;
    unicode[4934]:=16#8517;
    unicode[4935]:=16#851a;
    unicode[4936]:=16#851f;
    unicode[4937]:=16#8521;
    unicode[4938]:=16#852b;
    unicode[4939]:=16#852c;
    unicode[4940]:=16#8537;
    unicode[4941]:=16#8538;
    unicode[4942]:=16#8539;
    unicode[4943]:=16#853a;
    unicode[4944]:=16#853b;
    unicode[4945]:=16#853c;
    unicode[4946]:=16#853d;
    unicode[4947]:=16#8543;
    unicode[4948]:=16#8548;
    unicode[4949]:=16#8549;
    unicode[4950]:=16#854a;
    unicode[4951]:=16#8556;
    unicode[4952]:=16#8559;
    unicode[4953]:=16#855e;
    unicode[4954]:=16#8564;
    unicode[4955]:=16#8568;
    unicode[4956]:=16#8572;
    unicode[4957]:=16#8574;
    unicode[4958]:=16#8579;
    unicode[4959]:=16#857a;
    unicode[4960]:=16#857b;
    unicode[4961]:=16#857e;
    unicode[4962]:=16#8584;
    unicode[4963]:=16#8585;
    unicode[4964]:=16#8587;
    unicode[4965]:=16#858f;
    unicode[4966]:=16#859b;
    unicode[4967]:=16#859c;
    unicode[4968]:=16#85a4;
    unicode[4969]:=16#85a8;
    unicode[4970]:=16#85aa;
    unicode[4971]:=16#85ae;
    unicode[4972]:=16#85af;
    unicode[4973]:=16#85b0;
    unicode[4974]:=16#85b7;
    unicode[4975]:=16#85b9;
    unicode[4976]:=16#85c1;
    unicode[4977]:=16#85c9;
    unicode[4978]:=16#85cf;
    unicode[4979]:=16#85d0;
    unicode[4980]:=16#85d3;
    unicode[4981]:=16#85d5;
    unicode[4982]:=16#85dc;
    unicode[4983]:=16#85e4;
    unicode[4984]:=16#85e9;
    unicode[4985]:=16#85fb;
    unicode[4986]:=16#85ff;
    unicode[4987]:=16#8605;
    unicode[4988]:=16#8611;
    unicode[4989]:=16#8616;
    unicode[4990]:=16#8627;
    unicode[4991]:=16#8629;
    unicode[4992]:=16#8638;
    unicode[4993]:=16#863c;
    unicode[4994]:=16#864d;
    unicode[4995]:=16#864e;
    unicode[4996]:=16#864f;
    unicode[4997]:=16#8650;
    unicode[4998]:=16#8651;
    unicode[4999]:=16#8654;           //unicode码 4000-4999
END_IF;

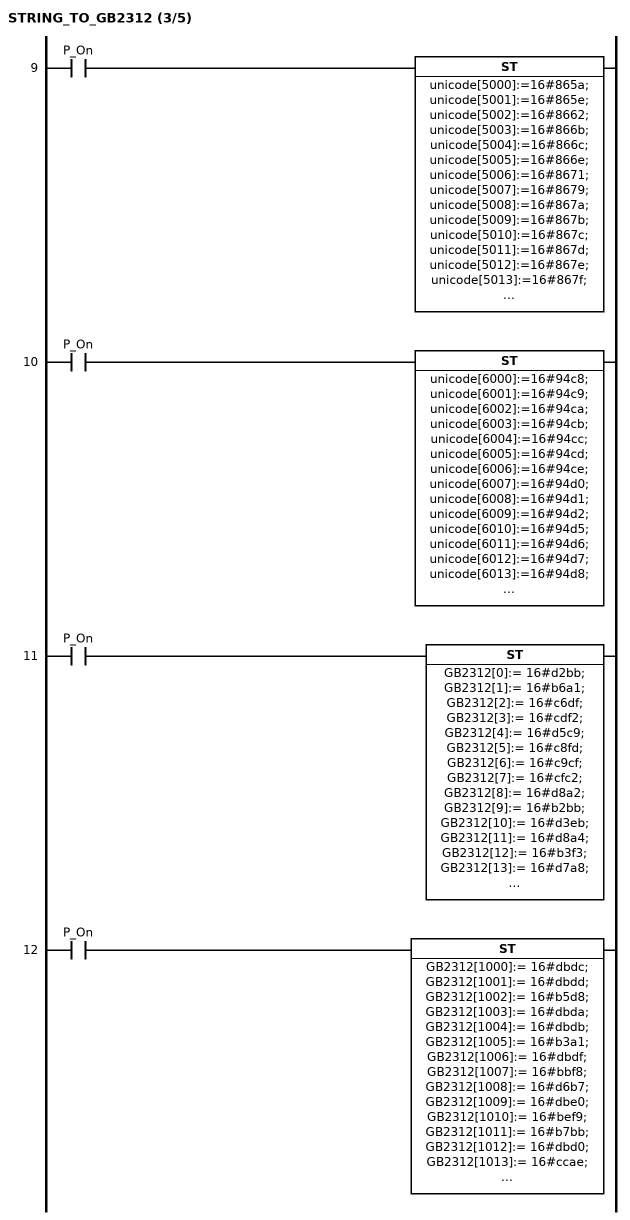
(* [picture p3: STRING_TO_GB2312, rungs 9-12] *)
(* Rung 9 *)
IF P_On THEN
    unicode[5000]:=16#865a;
    unicode[5001]:=16#865e;
    unicode[5002]:=16#8662;
    unicode[5003]:=16#866b;
    unicode[5004]:=16#866c;
    unicode[5005]:=16#866e;
    unicode[5006]:=16#8671;
    unicode[5007]:=16#8679;
    unicode[5008]:=16#867a;
    unicode[5009]:=16#867b;
    unicode[5010]:=16#867c;
    unicode[5011]:=16#867d;
    unicode[5012]:=16#867e;
    unicode[5013]:=16#867f;
    unicode[5014]:=16#8680;
    unicode[5015]:=16#8681;
    unicode[5016]:=16#8682;
    unicode[5017]:=16#868a;
    unicode[5018]:=16#868b;
    unicode[5019]:=16#868c;
    unicode[5020]:=16#868d;
    unicode[5021]:=16#8693;
    unicode[5022]:=16#8695;
    unicode[5023]:=16#869c;
    unicode[5024]:=16#869d;
    unicode[5025]:=16#86a3;
    unicode[5026]:=16#86a4;
    unicode[5027]:=16#86a7;
    unicode[5028]:=16#86a8;
    unicode[5029]:=16#86a9;
    unicode[5030]:=16#86aa;
    unicode[5031]:=16#86ac;
    unicode[5032]:=16#86af;
    unicode[5033]:=16#86b0;
    unicode[5034]:=16#86b1;
    unicode[5035]:=16#86b4;
    unicode[5036]:=16#86b5;
    unicode[5037]:=16#86b6;
    unicode[5038]:=16#86ba;
    unicode[5039]:=16#86c0;
    unicode[5040]:=16#86c4;
    unicode[5041]:=16#86c6;
    unicode[5042]:=16#86c7;
    unicode[5043]:=16#86c9;
    unicode[5044]:=16#86ca;
    unicode[5045]:=16#86cb;
    unicode[5046]:=16#86ce;
    unicode[5047]:=16#86cf;
    unicode[5048]:=16#86d0;
    unicode[5049]:=16#86d1;
    unicode[5050]:=16#86d4;
    unicode[5051]:=16#86d8;
    unicode[5052]:=16#86d9;
    unicode[5053]:=16#86db;
    unicode[5054]:=16#86de;
    unicode[5055]:=16#86df;
    unicode[5056]:=16#86e4;
    unicode[5057]:=16#86e9;
    unicode[5058]:=16#86ed;
    unicode[5059]:=16#86ee;
    unicode[5060]:=16#86f0;
    unicode[5061]:=16#86f1;
    unicode[5062]:=16#86f2;
    unicode[5063]:=16#86f3;
    unicode[5064]:=16#86f4;
    unicode[5065]:=16#86f8;
    unicode[5066]:=16#86f9;
    unicode[5067]:=16#86fe;
    unicode[5068]:=16#8700;
    unicode[5069]:=16#8702;
    unicode[5070]:=16#8703;
    unicode[5071]:=16#8707;
    unicode[5072]:=16#8708;
    unicode[5073]:=16#8709;
    unicode[5074]:=16#870a;
    unicode[5075]:=16#870d;
    unicode[5076]:=16#8712;
    unicode[5077]:=16#8713;
    unicode[5078]:=16#8715;
    unicode[5079]:=16#8717;
    unicode[5080]:=16#8718;
    unicode[5081]:=16#871a;
    unicode[5082]:=16#871c;
    unicode[5083]:=16#871e;
    unicode[5084]:=16#8721;
    unicode[5085]:=16#8722;
    unicode[5086]:=16#8723;
    unicode[5087]:=16#8725;
    unicode[5088]:=16#8729;
    unicode[5089]:=16#872e;
    unicode[5090]:=16#8731;
    unicode[5091]:=16#8734;
    unicode[5092]:=16#8737;
    unicode[5093]:=16#873b;
    unicode[5094]:=16#873e;
    unicode[5095]:=16#873f;
    unicode[5096]:=16#8747;
    unicode[5097]:=16#8748;
    unicode[5098]:=16#8749;
    unicode[5099]:=16#874c;
    unicode[5100]:=16#874e;
    unicode[5101]:=16#8753;
    unicode[5102]:=16#8757;
    unicode[5103]:=16#8759;
    unicode[5104]:=16#8760;
    unicode[5105]:=16#8763;
    unicode[5106]:=16#8764;
    unicode[5107]:=16#8765;
    unicode[5108]:=16#876e;
    unicode[5109]:=16#8770;
    unicode[5110]:=16#8774;
    unicode[5111]:=16#8776;
    unicode[5112]:=16#877b;
    unicode[5113]:=16#877c;
    unicode[5114]:=16#877d;
    unicode[5115]:=16#877e;
    unicode[5116]:=16#8782;
    unicode[5117]:=16#8783;
    unicode[5118]:=16#8785;
    unicode[5119]:=16#8788;
    unicode[5120]:=16#878b;
    unicode[5121]:=16#878d;
    unicode[5122]:=16#8793;
    unicode[5123]:=16#8797;
    unicode[5124]:=16#879f;
    unicode[5125]:=16#87a8;
    unicode[5126]:=16#87ab;
    unicode[5127]:=16#87ac;
    unicode[5128]:=16#87ad;
    unicode[5129]:=16#87af;
    unicode[5130]:=16#87b3;
    unicode[5131]:=16#87b5;
    unicode[5132]:=16#87ba;
    unicode[5133]:=16#87bd;
    unicode[5134]:=16#87c0;
    unicode[5135]:=16#87c6;
    unicode[5136]:=16#87ca;
    unicode[5137]:=16#87cb;
    unicode[5138]:=16#87d1;
    unicode[5139]:=16#87d2;
    unicode[5140]:=16#87d3;
    unicode[5141]:=16#87db;
    unicode[5142]:=16#87e0;
    unicode[5143]:=16#87e5;
    unicode[5144]:=16#87ea;
    unicode[5145]:=16#87ee;
    unicode[5146]:=16#87f9;
    unicode[5147]:=16#87fe;
    unicode[5148]:=16#8803;
    unicode[5149]:=16#880a;
    unicode[5150]:=16#8813;
    unicode[5151]:=16#8815;
    unicode[5152]:=16#8816;
    unicode[5153]:=16#881b;
    unicode[5154]:=16#8821;
    unicode[5155]:=16#8822;
    unicode[5156]:=16#8832;
    unicode[5157]:=16#8839;
    unicode[5158]:=16#883c;
    unicode[5159]:=16#8840;
    unicode[5160]:=16#8844;
    unicode[5161]:=16#8845;
    unicode[5162]:=16#884c;
    unicode[5163]:=16#884d;
    unicode[5164]:=16#8854;
    unicode[5165]:=16#8857;
    unicode[5166]:=16#8859;
    unicode[5167]:=16#8861;
    unicode[5168]:=16#8862;
    unicode[5169]:=16#8863;
    unicode[5170]:=16#8864;
    unicode[5171]:=16#8865;
    unicode[5172]:=16#8868;
    unicode[5173]:=16#8869;
    unicode[5174]:=16#886b;
    unicode[5175]:=16#886c;
    unicode[5176]:=16#886e;
    unicode[5177]:=16#8870;
    unicode[5178]:=16#8872;
    unicode[5179]:=16#8877;
    unicode[5180]:=16#887d;
    unicode[5181]:=16#887e;
    unicode[5182]:=16#887f;
    unicode[5183]:=16#8881;
    unicode[5184]:=16#8882;
    unicode[5185]:=16#8884;
    unicode[5186]:=16#8885;
    unicode[5187]:=16#8888;
    unicode[5188]:=16#888b;
    unicode[5189]:=16#888d;
    unicode[5190]:=16#8892;
    unicode[5191]:=16#8896;
    unicode[5192]:=16#889c;
    unicode[5193]:=16#88a2;
    unicode[5194]:=16#88a4;
    unicode[5195]:=16#88ab;
    unicode[5196]:=16#88ad;
    unicode[5197]:=16#88b1;
    unicode[5198]:=16#88b7;
    unicode[5199]:=16#88bc;
    unicode[5200]:=16#88c1;
    unicode[5201]:=16#88c2;
    unicode[5202]:=16#88c5;
    unicode[5203]:=16#88c6;
    unicode[5204]:=16#88c9;
    unicode[5205]:=16#88ce;
    unicode[5206]:=16#88d2;
    unicode[5207]:=16#88d4;
    unicode[5208]:=16#88d5;
    unicode[5209]:=16#88d8;
    unicode[5210]:=16#88d9;
    unicode[5211]:=16#88df;
    unicode[5212]:=16#88e2;
    unicode[5213]:=16#88e3;
    unicode[5214]:=16#88e4;
    unicode[5215]:=16#88e5;
    unicode[5216]:=16#88e8;
    unicode[5217]:=16#88f0;
    unicode[5218]:=16#88f1;
    unicode[5219]:=16#88f3;
    unicode[5220]:=16#88f4;
    unicode[5221]:=16#88f8;
    unicode[5222]:=16#88f9;
    unicode[5223]:=16#88fc;
    unicode[5224]:=16#88fe;
    unicode[5225]:=16#8902;
    unicode[5226]:=16#890a;
    unicode[5227]:=16#8910;
    unicode[5228]:=16#8912;
    unicode[5229]:=16#8913;
    unicode[5230]:=16#8919;
    unicode[5231]:=16#891a;
    unicode[5232]:=16#891b;
    unicode[5233]:=16#8921;
    unicode[5234]:=16#8925;
    unicode[5235]:=16#892a;
    unicode[5236]:=16#892b;
    unicode[5237]:=16#8930;
    unicode[5238]:=16#8934;
    unicode[5239]:=16#8936;
    unicode[5240]:=16#8941;
    unicode[5241]:=16#8944;
    unicode[5242]:=16#895e;
    unicode[5243]:=16#895f;
    unicode[5244]:=16#8966;
    unicode[5245]:=16#897b;
    unicode[5246]:=16#897f;
    unicode[5247]:=16#8981;
    unicode[5248]:=16#8983;
    unicode[5249]:=16#8986;
    unicode[5250]:=16#89c1;
    unicode[5251]:=16#89c2;
    unicode[5252]:=16#89c4;
    unicode[5253]:=16#89c5;
    unicode[5254]:=16#89c6;
    unicode[5255]:=16#89c7;
    unicode[5256]:=16#89c8;
    unicode[5257]:=16#89c9;
    unicode[5258]:=16#89ca;
    unicode[5259]:=16#89cb;
    unicode[5260]:=16#89cc;
    unicode[5261]:=16#89ce;
    unicode[5262]:=16#89cf;
    unicode[5263]:=16#89d0;
    unicode[5264]:=16#89d1;
    unicode[5265]:=16#89d2;
    unicode[5266]:=16#89d6;
    unicode[5267]:=16#89da;
    unicode[5268]:=16#89dc;
    unicode[5269]:=16#89de;
    unicode[5270]:=16#89e3;
    unicode[5271]:=16#89e5;
    unicode[5272]:=16#89e6;
    unicode[5273]:=16#89eb;
    unicode[5274]:=16#89ef;
    unicode[5275]:=16#89f3;
    unicode[5276]:=16#8a00;
    unicode[5277]:=16#8a07;
    unicode[5278]:=16#8a3e;
    unicode[5279]:=16#8a48;
    unicode[5280]:=16#8a79;
    unicode[5281]:=16#8a89;
    unicode[5282]:=16#8a8a;
    unicode[5283]:=16#8a93;
    unicode[5284]:=16#8b07;
    unicode[5285]:=16#8b26;
    unicode[5286]:=16#8b66;
    unicode[5287]:=16#8b6c;
    unicode[5288]:=16#8ba0;
    unicode[5289]:=16#8ba1;
    unicode[5290]:=16#8ba2;
    unicode[5291]:=16#8ba3;
    unicode[5292]:=16#8ba4;
    unicode[5293]:=16#8ba5;
    unicode[5294]:=16#8ba6;
    unicode[5295]:=16#8ba7;
    unicode[5296]:=16#8ba8;
    unicode[5297]:=16#8ba9;
    unicode[5298]:=16#8baa;
    unicode[5299]:=16#8bab;
    unicode[5300]:=16#8bad;
    unicode[5301]:=16#8bae;
    unicode[5302]:=16#8baf;
    unicode[5303]:=16#8bb0;
    unicode[5304]:=16#8bb2;
    unicode[5305]:=16#8bb3;
    unicode[5306]:=16#8bb4;
    unicode[5307]:=16#8bb5;
    unicode[5308]:=16#8bb6;
    unicode[5309]:=16#8bb7;
    unicode[5310]:=16#8bb8;
    unicode[5311]:=16#8bb9;
    unicode[5312]:=16#8bba;
    unicode[5313]:=16#8bbc;
    unicode[5314]:=16#8bbd;
    unicode[5315]:=16#8bbe;
    unicode[5316]:=16#8bbf;
    unicode[5317]:=16#8bc0;
    unicode[5318]:=16#8bc1;
    unicode[5319]:=16#8bc2;
    unicode[5320]:=16#8bc3;
    unicode[5321]:=16#8bc4;
    unicode[5322]:=16#8bc5;
    unicode[5323]:=16#8bc6;
    unicode[5324]:=16#8bc8;
    unicode[5325]:=16#8bc9;
    unicode[5326]:=16#8bca;
    unicode[5327]:=16#8bcb;
    unicode[5328]:=16#8bcc;
    unicode[5329]:=16#8bcd;
    unicode[5330]:=16#8bce;
    unicode[5331]:=16#8bcf;
    unicode[5332]:=16#8bd1;
    unicode[5333]:=16#8bd2;
    unicode[5334]:=16#8bd3;
    unicode[5335]:=16#8bd4;
    unicode[5336]:=16#8bd5;
    unicode[5337]:=16#8bd6;
    unicode[5338]:=16#8bd7;
    unicode[5339]:=16#8bd8;
    unicode[5340]:=16#8bd9;
    unicode[5341]:=16#8bda;
    unicode[5342]:=16#8bdb;
    unicode[5343]:=16#8bdc;
    unicode[5344]:=16#8bdd;
    unicode[5345]:=16#8bde;
    unicode[5346]:=16#8bdf;
    unicode[5347]:=16#8be0;
    unicode[5348]:=16#8be1;
    unicode[5349]:=16#8be2;
    unicode[5350]:=16#8be3;
    unicode[5351]:=16#8be4;
    unicode[5352]:=16#8be5;
    unicode[5353]:=16#8be6;
    unicode[5354]:=16#8be7;
    unicode[5355]:=16#8be8;
    unicode[5356]:=16#8be9;
    unicode[5357]:=16#8beb;
    unicode[5358]:=16#8bec;
    unicode[5359]:=16#8bed;
    unicode[5360]:=16#8bee;
    unicode[5361]:=16#8bef;
    unicode[5362]:=16#8bf0;
    unicode[5363]:=16#8bf1;
    unicode[5364]:=16#8bf2;
    unicode[5365]:=16#8bf3;
    unicode[5366]:=16#8bf4;
    unicode[5367]:=16#8bf5;
    unicode[5368]:=16#8bf6;
    unicode[5369]:=16#8bf7;
    unicode[5370]:=16#8bf8;
    unicode[5371]:=16#8bf9;
    unicode[5372]:=16#8bfa;
    unicode[5373]:=16#8bfb;
    unicode[5374]:=16#8bfc;
    unicode[5375]:=16#8bfd;
    unicode[5376]:=16#8bfe;
    unicode[5377]:=16#8bff;
    unicode[5378]:=16#8c00;
    unicode[5379]:=16#8c01;
    unicode[5380]:=16#8c02;
    unicode[5381]:=16#8c03;
    unicode[5382]:=16#8c04;
    unicode[5383]:=16#8c05;
    unicode[5384]:=16#8c06;
    unicode[5385]:=16#8c07;
    unicode[5386]:=16#8c08;
    unicode[5387]:=16#8c0a;
    unicode[5388]:=16#8c0b;
    unicode[5389]:=16#8c0c;
    unicode[5390]:=16#8c0d;
    unicode[5391]:=16#8c0e;
    unicode[5392]:=16#8c0f;
    unicode[5393]:=16#8c10;
    unicode[5394]:=16#8c11;
    unicode[5395]:=16#8c12;
    unicode[5396]:=16#8c13;
    unicode[5397]:=16#8c14;
    unicode[5398]:=16#8c15;
    unicode[5399]:=16#8c16;
    unicode[5400]:=16#8c17;
    unicode[5401]:=16#8c18;
    unicode[5402]:=16#8c19;
    unicode[5403]:=16#8c1a;
    unicode[5404]:=16#8c1b;
    unicode[5405]:=16#8c1c;
    unicode[5406]:=16#8c1d;
    unicode[5407]:=16#8c1f;
    unicode[5408]:=16#8c20;
    unicode[5409]:=16#8c21;
    unicode[5410]:=16#8c22;
    unicode[5411]:=16#8c23;
    unicode[5412]:=16#8c24;
    unicode[5413]:=16#8c25;
    unicode[5414]:=16#8c26;
    unicode[5415]:=16#8c27;
    unicode[5416]:=16#8c28;
    unicode[5417]:=16#8c29;
    unicode[5418]:=16#8c2a;
    unicode[5419]:=16#8c2b;
    unicode[5420]:=16#8c2c;
    unicode[5421]:=16#8c2d;
    unicode[5422]:=16#8c2e;
    unicode[5423]:=16#8c2f;
    unicode[5424]:=16#8c30;
    unicode[5425]:=16#8c31;
    unicode[5426]:=16#8c32;
    unicode[5427]:=16#8c33;
    unicode[5428]:=16#8c34;
    unicode[5429]:=16#8c35;
    unicode[5430]:=16#8c36;
    unicode[5431]:=16#8c37;
    unicode[5432]:=16#8c41;
    unicode[5433]:=16#8c46;
    unicode[5434]:=16#8c47;
    unicode[5435]:=16#8c49;
    unicode[5436]:=16#8c4c;
    unicode[5437]:=16#8c55;
    unicode[5438]:=16#8c5a;
    unicode[5439]:=16#8c61;
    unicode[5440]:=16#8c62;
    unicode[5441]:=16#8c6a;
    unicode[5442]:=16#8c6b;
    unicode[5443]:=16#8c73;
    unicode[5444]:=16#8c78;
    unicode[5445]:=16#8c79;
    unicode[5446]:=16#8c7a;
    unicode[5447]:=16#8c82;
    unicode[5448]:=16#8c85;
    unicode[5449]:=16#8c89;
    unicode[5450]:=16#8c8a;
    unicode[5451]:=16#8c8c;
    unicode[5452]:=16#8c94;
    unicode[5453]:=16#8c98;
    unicode[5454]:=16#8d1d;
    unicode[5455]:=16#8d1e;
    unicode[5456]:=16#8d1f;
    unicode[5457]:=16#8d21;
    unicode[5458]:=16#8d22;
    unicode[5459]:=16#8d23;
    unicode[5460]:=16#8d24;
    unicode[5461]:=16#8d25;
    unicode[5462]:=16#8d26;
    unicode[5463]:=16#8d27;
    unicode[5464]:=16#8d28;
    unicode[5465]:=16#8d29;
    unicode[5466]:=16#8d2a;
    unicode[5467]:=16#8d2b;
    unicode[5468]:=16#8d2c;
    unicode[5469]:=16#8d2d;
    unicode[5470]:=16#8d2e;
    unicode[5471]:=16#8d2f;
    unicode[5472]:=16#8d30;
    unicode[5473]:=16#8d31;
    unicode[5474]:=16#8d32;
    unicode[5475]:=16#8d33;
    unicode[5476]:=16#8d34;
    unicode[5477]:=16#8d35;
    unicode[5478]:=16#8d36;
    unicode[5479]:=16#8d37;
    unicode[5480]:=16#8d38;
    unicode[5481]:=16#8d39;
    unicode[5482]:=16#8d3a;
    unicode[5483]:=16#8d3b;
    unicode[5484]:=16#8d3c;
    unicode[5485]:=16#8d3d;
    unicode[5486]:=16#8d3e;
    unicode[5487]:=16#8d3f;
    unicode[5488]:=16#8d40;
    unicode[5489]:=16#8d41;
    unicode[5490]:=16#8d42;
    unicode[5491]:=16#8d43;
    unicode[5492]:=16#8d44;
    unicode[5493]:=16#8d45;
    unicode[5494]:=16#8d46;
    unicode[5495]:=16#8d47;
    unicode[5496]:=16#8d48;
    unicode[5497]:=16#8d49;
    unicode[5498]:=16#8d4a;
    unicode[5499]:=16#8d4b;
    unicode[5500]:=16#8d4c;
    unicode[5501]:=16#8d4d;
    unicode[5502]:=16#8d4e;
    unicode[5503]:=16#8d4f;
    unicode[5504]:=16#8d50;
    unicode[5505]:=16#8d53;
    unicode[5506]:=16#8d54;
    unicode[5507]:=16#8d55;
    unicode[5508]:=16#8d56;
    unicode[5509]:=16#8d58;
    unicode[5510]:=16#8d59;
    unicode[5511]:=16#8d5a;
    unicode[5512]:=16#8d5b;
    unicode[5513]:=16#8d5c;
    unicode[5514]:=16#8d5d;
    unicode[5515]:=16#8d5e;
    unicode[5516]:=16#8d60;
    unicode[5517]:=16#8d61;
    unicode[5518]:=16#8d62;
    unicode[5519]:=16#8d63;
    unicode[5520]:=16#8d64;
    unicode[5521]:=16#8d66;
    unicode[5522]:=16#8d67;
    unicode[5523]:=16#8d6b;
    unicode[5524]:=16#8d6d;
    unicode[5525]:=16#8d70;
    unicode[5526]:=16#8d73;
    unicode[5527]:=16#8d74;
    unicode[5528]:=16#8d75;
    unicode[5529]:=16#8d76;
    unicode[5530]:=16#8d77;
    unicode[5531]:=16#8d81;
    unicode[5532]:=16#8d84;
    unicode[5533]:=16#8d85;
    unicode[5534]:=16#8d8a;
    unicode[5535]:=16#8d8b;
    unicode[5536]:=16#8d91;
    unicode[5537]:=16#8d94;
    unicode[5538]:=16#8d9f;
    unicode[5539]:=16#8da3;
    unicode[5540]:=16#8db1;
    unicode[5541]:=16#8db3;
    unicode[5542]:=16#8db4;
    unicode[5543]:=16#8db5;
    unicode[5544]:=16#8db8;
    unicode[5545]:=16#8dba;
    unicode[5546]:=16#8dbc;
    unicode[5547]:=16#8dbe;
    unicode[5548]:=16#8dbf;
    unicode[5549]:=16#8dc3;
    unicode[5550]:=16#8dc4;
    unicode[5551]:=16#8dc6;
    unicode[5552]:=16#8dcb;
    unicode[5553]:=16#8dcc;
    unicode[5554]:=16#8dce;
    unicode[5555]:=16#8dcf;
    unicode[5556]:=16#8dd1;
    unicode[5557]:=16#8dd6;
    unicode[5558]:=16#8dd7;
    unicode[5559]:=16#8dda;
    unicode[5560]:=16#8ddb;
    unicode[5561]:=16#8ddd;
    unicode[5562]:=16#8dde;
    unicode[5563]:=16#8ddf;
    unicode[5564]:=16#8de3;
    unicode[5565]:=16#8de4;
    unicode[5566]:=16#8de8;
    unicode[5567]:=16#8dea;
    unicode[5568]:=16#8deb;
    unicode[5569]:=16#8dec;
    unicode[5570]:=16#8def;
    unicode[5571]:=16#8df3;
    unicode[5572]:=16#8df5;
    unicode[5573]:=16#8df7;
    unicode[5574]:=16#8df8;
    unicode[5575]:=16#8df9;
    unicode[5576]:=16#8dfa;
    unicode[5577]:=16#8dfb;
    unicode[5578]:=16#8dfd;
    unicode[5579]:=16#8e05;
    unicode[5580]:=16#8e09;
    unicode[5581]:=16#8e0a;
    unicode[5582]:=16#8e0c;
    unicode[5583]:=16#8e0f;
    unicode[5584]:=16#8e14;
    unicode[5585]:=16#8e1d;
    unicode[5586]:=16#8e1e;
    unicode[5587]:=16#8e1f;
    unicode[5588]:=16#8e22;
    unicode[5589]:=16#8e23;
    unicode[5590]:=16#8e29;
    unicode[5591]:=16#8e2a;
    unicode[5592]:=16#8e2c;
    unicode[5593]:=16#8e2e;
    unicode[5594]:=16#8e2f;
    unicode[5595]:=16#8e31;
    unicode[5596]:=16#8e35;
    unicode[5597]:=16#8e39;
    unicode[5598]:=16#8e3a;
    unicode[5599]:=16#8e3d;
    unicode[5600]:=16#8e40;
    unicode[5601]:=16#8e41;
    unicode[5602]:=16#8e42;
    unicode[5603]:=16#8e44;
    unicode[5604]:=16#8e47;
    unicode[5605]:=16#8e48;
    unicode[5606]:=16#8e49;
    unicode[5607]:=16#8e4a;
    unicode[5608]:=16#8e4b;
    unicode[5609]:=16#8e51;
    unicode[5610]:=16#8e52;
    unicode[5611]:=16#8e59;
    unicode[5612]:=16#8e66;
    unicode[5613]:=16#8e69;
    unicode[5614]:=16#8e6c;
    unicode[5615]:=16#8e6d;
    unicode[5616]:=16#8e6f;
    unicode[5617]:=16#8e70;
    unicode[5618]:=16#8e72;
    unicode[5619]:=16#8e74;
    unicode[5620]:=16#8e76;
    unicode[5621]:=16#8e7c;
    unicode[5622]:=16#8e7f;
    unicode[5623]:=16#8e81;
    unicode[5624]:=16#8e85;
    unicode[5625]:=16#8e87;
    unicode[5626]:=16#8e8f;
    unicode[5627]:=16#8e90;
    unicode[5628]:=16#8e94;
    unicode[5629]:=16#8e9c;
    unicode[5630]:=16#8e9e;
    unicode[5631]:=16#8eab;
    unicode[5632]:=16#8eac;
    unicode[5633]:=16#8eaf;
    unicode[5634]:=16#8eb2;
    unicode[5635]:=16#8eba;
    unicode[5636]:=16#8ece;
    unicode[5637]:=16#8f66;
    unicode[5638]:=16#8f67;
    unicode[5639]:=16#8f68;
    unicode[5640]:=16#8f69;
    unicode[5641]:=16#8f6b;
    unicode[5642]:=16#8f6c;
    unicode[5643]:=16#8f6d;
    unicode[5644]:=16#8f6e;
    unicode[5645]:=16#8f6f;
    unicode[5646]:=16#8f70;
    unicode[5647]:=16#8f71;
    unicode[5648]:=16#8f72;
    unicode[5649]:=16#8f73;
    unicode[5650]:=16#8f74;
    unicode[5651]:=16#8f75;
    unicode[5652]:=16#8f76;
    unicode[5653]:=16#8f77;
    unicode[5654]:=16#8f78;
    unicode[5655]:=16#8f79;
    unicode[5656]:=16#8f7a;
    unicode[5657]:=16#8f7b;
    unicode[5658]:=16#8f7c;
    unicode[5659]:=16#8f7d;
    unicode[5660]:=16#8f7e;
    unicode[5661]:=16#8f7f;
    unicode[5662]:=16#8f81;
    unicode[5663]:=16#8f82;
    unicode[5664]:=16#8f83;
    unicode[5665]:=16#8f84;
    unicode[5666]:=16#8f85;
    unicode[5667]:=16#8f86;
    unicode[5668]:=16#8f87;
    unicode[5669]:=16#8f88;
    unicode[5670]:=16#8f89;
    unicode[5671]:=16#8f8a;
    unicode[5672]:=16#8f8b;
    unicode[5673]:=16#8f8d;
    unicode[5674]:=16#8f8e;
    unicode[5675]:=16#8f8f;
    unicode[5676]:=16#8f90;
    unicode[5677]:=16#8f91;
    unicode[5678]:=16#8f93;
    unicode[5679]:=16#8f94;
    unicode[5680]:=16#8f95;
    unicode[5681]:=16#8f96;
    unicode[5682]:=16#8f97;
    unicode[5683]:=16#8f98;
    unicode[5684]:=16#8f99;
    unicode[5685]:=16#8f9a;
    unicode[5686]:=16#8f9b;
    unicode[5687]:=16#8f9c;
    unicode[5688]:=16#8f9e;
    unicode[5689]:=16#8f9f;
    unicode[5690]:=16#8fa3;
    unicode[5691]:=16#8fa8;
    unicode[5692]:=16#8fa9;
    unicode[5693]:=16#8fab;
    unicode[5694]:=16#8fb0;
    unicode[5695]:=16#8fb1;
    unicode[5696]:=16#8fb6;
    unicode[5697]:=16#8fb9;
    unicode[5698]:=16#8fbd;
    unicode[5699]:=16#8fbe;
    unicode[5700]:=16#8fc1;
    unicode[5701]:=16#8fc2;
    unicode[5702]:=16#8fc4;
    unicode[5703]:=16#8fc5;
    unicode[5704]:=16#8fc7;
    unicode[5705]:=16#8fc8;
    unicode[5706]:=16#8fce;
    unicode[5707]:=16#8fd0;
    unicode[5708]:=16#8fd1;
    unicode[5709]:=16#8fd3;
    unicode[5710]:=16#8fd4;
    unicode[5711]:=16#8fd5;
    unicode[5712]:=16#8fd8;
    unicode[5713]:=16#8fd9;
    unicode[5714]:=16#8fdb;
    unicode[5715]:=16#8fdc;
    unicode[5716]:=16#8fdd;
    unicode[5717]:=16#8fde;
    unicode[5718]:=16#8fdf;
    unicode[5719]:=16#8fe2;
    unicode[5720]:=16#8fe4;
    unicode[5721]:=16#8fe5;
    unicode[5722]:=16#8fe6;
    unicode[5723]:=16#8fe8;
    unicode[5724]:=16#8fe9;
    unicode[5725]:=16#8fea;
    unicode[5726]:=16#8feb;
    unicode[5727]:=16#8fed;
    unicode[5728]:=16#8fee;
    unicode[5729]:=16#8ff0;
    unicode[5730]:=16#8ff3;
    unicode[5731]:=16#8ff7;
    unicode[5732]:=16#8ff8;
    unicode[5733]:=16#8ff9;
    unicode[5734]:=16#8ffd;
    unicode[5735]:=16#9000;
    unicode[5736]:=16#9001;
    unicode[5737]:=16#9002;
    unicode[5738]:=16#9003;
    unicode[5739]:=16#9004;
    unicode[5740]:=16#9005;
    unicode[5741]:=16#9006;
    unicode[5742]:=16#9009;
    unicode[5743]:=16#900a;
    unicode[5744]:=16#900b;
    unicode[5745]:=16#900d;
    unicode[5746]:=16#900f;
    unicode[5747]:=16#9010;
    unicode[5748]:=16#9011;
    unicode[5749]:=16#9012;
    unicode[5750]:=16#9014;
    unicode[5751]:=16#9016;
    unicode[5752]:=16#9017;
    unicode[5753]:=16#901a;
    unicode[5754]:=16#901b;
    unicode[5755]:=16#901d;
    unicode[5756]:=16#901e;
    unicode[5757]:=16#901f;
    unicode[5758]:=16#9020;
    unicode[5759]:=16#9021;
    unicode[5760]:=16#9022;
    unicode[5761]:=16#9026;
    unicode[5762]:=16#902d;
    unicode[5763]:=16#902e;
    unicode[5764]:=16#902f;
    unicode[5765]:=16#9035;
    unicode[5766]:=16#9036;
    unicode[5767]:=16#9038;
    unicode[5768]:=16#903b;
    unicode[5769]:=16#903c;
    unicode[5770]:=16#903e;
    unicode[5771]:=16#9041;
    unicode[5772]:=16#9042;
    unicode[5773]:=16#9044;
    unicode[5774]:=16#9047;
    unicode[5775]:=16#904d;
    unicode[5776]:=16#904f;
    unicode[5777]:=16#9050;
    unicode[5778]:=16#9051;
    unicode[5779]:=16#9052;
    unicode[5780]:=16#9053;
    unicode[5781]:=16#9057;
    unicode[5782]:=16#9058;
    unicode[5783]:=16#905b;
    unicode[5784]:=16#9062;
    unicode[5785]:=16#9063;
    unicode[5786]:=16#9065;
    unicode[5787]:=16#9068;
    unicode[5788]:=16#906d;
    unicode[5789]:=16#906e;
    unicode[5790]:=16#9074;
    unicode[5791]:=16#9075;
    unicode[5792]:=16#907d;
    unicode[5793]:=16#907f;
    unicode[5794]:=16#9080;
    unicode[5795]:=16#9082;
    unicode[5796]:=16#9083;
    unicode[5797]:=16#9088;
    unicode[5798]:=16#908b;
    unicode[5799]:=16#9091;
    unicode[5800]:=16#9093;
    unicode[5801]:=16#9095;
    unicode[5802]:=16#9097;
    unicode[5803]:=16#9099;
    unicode[5804]:=16#909b;
    unicode[5805]:=16#909d;
    unicode[5806]:=16#90a1;
    unicode[5807]:=16#90a2;
    unicode[5808]:=16#90a3;
    unicode[5809]:=16#90a6;
    unicode[5810]:=16#90aa;
    unicode[5811]:=16#90ac;
    unicode[5812]:=16#90ae;
    unicode[5813]:=16#90af;
    unicode[5814]:=16#90b0;
    unicode[5815]:=16#90b1;
    unicode[5816]:=16#90b3;
    unicode[5817]:=16#90b4;
    unicode[5818]:=16#90b5;
    unicode[5819]:=16#90b6;
    unicode[5820]:=16#90b8;
    unicode[5821]:=16#90b9;
    unicode[5822]:=16#90ba;
    unicode[5823]:=16#90bb;
    unicode[5824]:=16#90be;
    unicode[5825]:=16#90c1;
    unicode[5826]:=16#90c4;
    unicode[5827]:=16#90c5;
    unicode[5828]:=16#90c7;
    unicode[5829]:=16#90ca;
    unicode[5830]:=16#90ce;
    unicode[5831]:=16#90cf;
    unicode[5832]:=16#90d0;
    unicode[5833]:=16#90d1;
    unicode[5834]:=16#90d3;
    unicode[5835]:=16#90d7;
    unicode[5836]:=16#90db;
    unicode[5837]:=16#90dc;
    unicode[5838]:=16#90dd;
    unicode[5839]:=16#90e1;
    unicode[5840]:=16#90e2;
    unicode[5841]:=16#90e6;
    unicode[5842]:=16#90e7;
    unicode[5843]:=16#90e8;
    unicode[5844]:=16#90eb;
    unicode[5845]:=16#90ed;
    unicode[5846]:=16#90ef;
    unicode[5847]:=16#90f4;
    unicode[5848]:=16#90f8;
    unicode[5849]:=16#90fd;
    unicode[5850]:=16#90fe;
    unicode[5851]:=16#9102;
    unicode[5852]:=16#9104;
    unicode[5853]:=16#9119;
    unicode[5854]:=16#911e;
    unicode[5855]:=16#9122;
    unicode[5856]:=16#9123;
    unicode[5857]:=16#912f;
    unicode[5858]:=16#9131;
    unicode[5859]:=16#9139;
    unicode[5860]:=16#9143;
    unicode[5861]:=16#9146;
    unicode[5862]:=16#9149;
    unicode[5863]:=16#914a;
    unicode[5864]:=16#914b;
    unicode[5865]:=16#914c;
    unicode[5866]:=16#914d;
    unicode[5867]:=16#914e;
    unicode[5868]:=16#914f;
    unicode[5869]:=16#9150;
    unicode[5870]:=16#9152;
    unicode[5871]:=16#9157;
    unicode[5872]:=16#915a;
    unicode[5873]:=16#915d;
    unicode[5874]:=16#915e;
    unicode[5875]:=16#9161;
    unicode[5876]:=16#9162;
    unicode[5877]:=16#9163;
    unicode[5878]:=16#9164;
    unicode[5879]:=16#9165;
    unicode[5880]:=16#9169;
    unicode[5881]:=16#916a;
    unicode[5882]:=16#916c;
    unicode[5883]:=16#916e;
    unicode[5884]:=16#916f;
    unicode[5885]:=16#9170;
    unicode[5886]:=16#9171;
    unicode[5887]:=16#9172;
    unicode[5888]:=16#9174;
    unicode[5889]:=16#9175;
    unicode[5890]:=16#9176;
    unicode[5891]:=16#9177;
    unicode[5892]:=16#9178;
    unicode[5893]:=16#9179;
    unicode[5894]:=16#917d;
    unicode[5895]:=16#917e;
    unicode[5896]:=16#917f;
    unicode[5897]:=16#9185;
    unicode[5898]:=16#9187;
    unicode[5899]:=16#9189;
    unicode[5900]:=16#918b;
    unicode[5901]:=16#918c;
    unicode[5902]:=16#918d;
    unicode[5903]:=16#9190;
    unicode[5904]:=16#9191;
    unicode[5905]:=16#9192;
    unicode[5906]:=16#919a;
    unicode[5907]:=16#919b;
    unicode[5908]:=16#91a2;
    unicode[5909]:=16#91a3;
    unicode[5910]:=16#91aa;
    unicode[5911]:=16#91ad;
    unicode[5912]:=16#91ae;
    unicode[5913]:=16#91af;
    unicode[5914]:=16#91b4;
    unicode[5915]:=16#91b5;
    unicode[5916]:=16#91ba;
    unicode[5917]:=16#91c7;
    unicode[5918]:=16#91c9;
    unicode[5919]:=16#91ca;
    unicode[5920]:=16#91cc;
    unicode[5921]:=16#91cd;
    unicode[5922]:=16#91ce;
    unicode[5923]:=16#91cf;
    unicode[5924]:=16#91d1;
    unicode[5925]:=16#91dc;
    unicode[5926]:=16#9274;
    unicode[5927]:=16#928e;
    unicode[5928]:=16#92ae;
    unicode[5929]:=16#92c8;
    unicode[5930]:=16#933e;
    unicode[5931]:=16#936a;
    unicode[5932]:=16#938f;
    unicode[5933]:=16#93ca;
    unicode[5934]:=16#93d6;
    unicode[5935]:=16#943e;
    unicode[5936]:=16#946b;
    unicode[5937]:=16#9485;
    unicode[5938]:=16#9486;
    unicode[5939]:=16#9487;
    unicode[5940]:=16#9488;
    unicode[5941]:=16#9489;
    unicode[5942]:=16#948a;
    unicode[5943]:=16#948b;
    unicode[5944]:=16#948c;
    unicode[5945]:=16#948d;
    unicode[5946]:=16#948e;
    unicode[5947]:=16#948f;
    unicode[5948]:=16#9490;
    unicode[5949]:=16#9492;
    unicode[5950]:=16#9493;
    unicode[5951]:=16#9494;
    unicode[5952]:=16#9495;
    unicode[5953]:=16#9497;
    unicode[5954]:=16#9499;
    unicode[5955]:=16#949a;
    unicode[5956]:=16#949b;
    unicode[5957]:=16#949c;
    unicode[5958]:=16#949d;
    unicode[5959]:=16#949e;
    unicode[5960]:=16#949f;
    unicode[5961]:=16#94a0;
    unicode[5962]:=16#94a1;
    unicode[5963]:=16#94a2;
    unicode[5964]:=16#94a3;
    unicode[5965]:=16#94a4;
    unicode[5966]:=16#94a5;
    unicode[5967]:=16#94a6;
    unicode[5968]:=16#94a7;
    unicode[5969]:=16#94a8;
    unicode[5970]:=16#94a9;
    unicode[5971]:=16#94aa;
    unicode[5972]:=16#94ab;
    unicode[5973]:=16#94ac;
    unicode[5974]:=16#94ad;
    unicode[5975]:=16#94ae;
    unicode[5976]:=16#94af;
    unicode[5977]:=16#94b0;
    unicode[5978]:=16#94b1;
    unicode[5979]:=16#94b2;
    unicode[5980]:=16#94b3;
    unicode[5981]:=16#94b4;
    unicode[5982]:=16#94b5;
    unicode[5983]:=16#94b6;
    unicode[5984]:=16#94b7;
    unicode[5985]:=16#94b8;
    unicode[5986]:=16#94b9;
    unicode[5987]:=16#94ba;
    unicode[5988]:=16#94bb;
    unicode[5989]:=16#94bc;
    unicode[5990]:=16#94bd;
    unicode[5991]:=16#94be;
    unicode[5992]:=16#94bf;
    unicode[5993]:=16#94c0;
    unicode[5994]:=16#94c1;
    unicode[5995]:=16#94c2;
    unicode[5996]:=16#94c3;
    unicode[5997]:=16#94c4;
    unicode[5998]:=16#94c5;
    unicode[5999]:=16#94c6;             //unicode码 5000-5999
END_IF;
(* Rung 10 *)
IF P_On THEN
    unicode[6000]:=16#94c8;
    unicode[6001]:=16#94c9;
    unicode[6002]:=16#94ca;
    unicode[6003]:=16#94cb;
    unicode[6004]:=16#94cc;
    unicode[6005]:=16#94cd;
    unicode[6006]:=16#94ce;
    unicode[6007]:=16#94d0;
    unicode[6008]:=16#94d1;
    unicode[6009]:=16#94d2;
    unicode[6010]:=16#94d5;
    unicode[6011]:=16#94d6;
    unicode[6012]:=16#94d7;
    unicode[6013]:=16#94d8;
    unicode[6014]:=16#94d9;
    unicode[6015]:=16#94db;
    unicode[6016]:=16#94dc;
    unicode[6017]:=16#94dd;
    unicode[6018]:=16#94de;
    unicode[6019]:=16#94df;
    unicode[6020]:=16#94e0;
    unicode[6021]:=16#94e1;
    unicode[6022]:=16#94e2;
    unicode[6023]:=16#94e3;
    unicode[6024]:=16#94e4;
    unicode[6025]:=16#94e5;
    unicode[6026]:=16#94e7;
    unicode[6027]:=16#94e8;
    unicode[6028]:=16#94e9;
    unicode[6029]:=16#94ea;
    unicode[6030]:=16#94eb;
    unicode[6031]:=16#94ec;
    unicode[6032]:=16#94ed;
    unicode[6033]:=16#94ee;
    unicode[6034]:=16#94ef;
    unicode[6035]:=16#94f0;
    unicode[6036]:=16#94f1;
    unicode[6037]:=16#94f2;
    unicode[6038]:=16#94f3;
    unicode[6039]:=16#94f4;
    unicode[6040]:=16#94f5;
    unicode[6041]:=16#94f6;
    unicode[6042]:=16#94f7;
    unicode[6043]:=16#94f8;
    unicode[6044]:=16#94f9;
    unicode[6045]:=16#94fa;
    unicode[6046]:=16#94fc;
    unicode[6047]:=16#94fd;
    unicode[6048]:=16#94fe;
    unicode[6049]:=16#94ff;
    unicode[6050]:=16#9500;
    unicode[6051]:=16#9501;
    unicode[6052]:=16#9502;
    unicode[6053]:=16#9503;
    unicode[6054]:=16#9504;
    unicode[6055]:=16#9505;
    unicode[6056]:=16#9506;
    unicode[6057]:=16#9507;
    unicode[6058]:=16#9508;
    unicode[6059]:=16#9509;
    unicode[6060]:=16#950a;
    unicode[6061]:=16#950b;
    unicode[6062]:=16#950c;
    unicode[6063]:=16#950d;
    unicode[6064]:=16#950e;
    unicode[6065]:=16#950f;
    unicode[6066]:=16#9510;
    unicode[6067]:=16#9511;
    unicode[6068]:=16#9512;
    unicode[6069]:=16#9513;
    unicode[6070]:=16#9514;
    unicode[6071]:=16#9515;
    unicode[6072]:=16#9516;
    unicode[6073]:=16#9517;
    unicode[6074]:=16#9518;
    unicode[6075]:=16#9519;
    unicode[6076]:=16#951a;
    unicode[6077]:=16#951b;
    unicode[6078]:=16#951d;
    unicode[6079]:=16#951e;
    unicode[6080]:=16#951f;
    unicode[6081]:=16#9521;
    unicode[6082]:=16#9522;
    unicode[6083]:=16#9523;
    unicode[6084]:=16#9524;
    unicode[6085]:=16#9525;
    unicode[6086]:=16#9526;
    unicode[6087]:=16#9528;
    unicode[6088]:=16#9529;
    unicode[6089]:=16#952a;
    unicode[6090]:=16#952b;
    unicode[6091]:=16#952c;
    unicode[6092]:=16#952d;
    unicode[6093]:=16#952e;
    unicode[6094]:=16#952f;
    unicode[6095]:=16#9530;
    unicode[6096]:=16#9531;
    unicode[6097]:=16#9532;
    unicode[6098]:=16#9534;
    unicode[6099]:=16#9535;
    unicode[6100]:=16#9536;
    unicode[6101]:=16#9537;
    unicode[6102]:=16#9538;
    unicode[6103]:=16#9539;
    unicode[6104]:=16#953a;
    unicode[6105]:=16#953b;
    unicode[6106]:=16#953c;
    unicode[6107]:=16#953e;
    unicode[6108]:=16#953f;
    unicode[6109]:=16#9540;
    unicode[6110]:=16#9541;
    unicode[6111]:=16#9542;
    unicode[6112]:=16#9544;
    unicode[6113]:=16#9545;
    unicode[6114]:=16#9546;
    unicode[6115]:=16#9547;
    unicode[6116]:=16#9549;
    unicode[6117]:=16#954a;
    unicode[6118]:=16#954c;
    unicode[6119]:=16#954d;
    unicode[6120]:=16#954e;
    unicode[6121]:=16#954f;
    unicode[6122]:=16#9550;
    unicode[6123]:=16#9551;
    unicode[6124]:=16#9552;
    unicode[6125]:=16#9553;
    unicode[6126]:=16#9554;
    unicode[6127]:=16#9556;
    unicode[6128]:=16#9557;
    unicode[6129]:=16#9558;
    unicode[6130]:=16#9559;
    unicode[6131]:=16#955b;
    unicode[6132]:=16#955c;
    unicode[6133]:=16#955d;
    unicode[6134]:=16#955e;
    unicode[6135]:=16#955f;
    unicode[6136]:=16#9561;
    unicode[6137]:=16#9562;
    unicode[6138]:=16#9563;
    unicode[6139]:=16#9564;
    unicode[6140]:=16#9565;
    unicode[6141]:=16#9566;
    unicode[6142]:=16#9567;
    unicode[6143]:=16#9568;
    unicode[6144]:=16#9569;
    unicode[6145]:=16#956a;
    unicode[6146]:=16#956b;
    unicode[6147]:=16#956c;
    unicode[6148]:=16#956d;
    unicode[6149]:=16#956f;
    unicode[6150]:=16#9570;
    unicode[6151]:=16#9571;
    unicode[6152]:=16#9572;
    unicode[6153]:=16#9573;
    unicode[6154]:=16#9576;
    unicode[6155]:=16#957f;
    unicode[6156]:=16#95e8;
    unicode[6157]:=16#95e9;
    unicode[6158]:=16#95ea;
    unicode[6159]:=16#95eb;
    unicode[6160]:=16#95ed;
    unicode[6161]:=16#95ee;
    unicode[6162]:=16#95ef;
    unicode[6163]:=16#95f0;
    unicode[6164]:=16#95f1;
    unicode[6165]:=16#95f2;
    unicode[6166]:=16#95f3;
    unicode[6167]:=16#95f4;
    unicode[6168]:=16#95f5;
    unicode[6169]:=16#95f6;
    unicode[6170]:=16#95f7;
    unicode[6171]:=16#95f8;
    unicode[6172]:=16#95f9;
    unicode[6173]:=16#95fa;
    unicode[6174]:=16#95fb;
    unicode[6175]:=16#95fc;
    unicode[6176]:=16#95fd;
    unicode[6177]:=16#95fe;
    unicode[6178]:=16#9600;
    unicode[6179]:=16#9601;
    unicode[6180]:=16#9602;
    unicode[6181]:=16#9603;
    unicode[6182]:=16#9604;
    unicode[6183]:=16#9605;
    unicode[6184]:=16#9606;
    unicode[6185]:=16#9608;
    unicode[6186]:=16#9609;
    unicode[6187]:=16#960a;
    unicode[6188]:=16#960b;
    unicode[6189]:=16#960c;
    unicode[6190]:=16#960d;
    unicode[6191]:=16#960e;
    unicode[6192]:=16#960f;
    unicode[6193]:=16#9610;
    unicode[6194]:=16#9611;
    unicode[6195]:=16#9612;
    unicode[6196]:=16#9614;
    unicode[6197]:=16#9615;
    unicode[6198]:=16#9616;
    unicode[6199]:=16#9617;
    unicode[6200]:=16#9619;
    unicode[6201]:=16#961a;
    unicode[6202]:=16#961c;
    unicode[6203]:=16#961d;
    unicode[6204]:=16#961f;
    unicode[6205]:=16#9621;
    unicode[6206]:=16#9622;
    unicode[6207]:=16#962a;
    unicode[6208]:=16#962e;
    unicode[6209]:=16#9631;
    unicode[6210]:=16#9632;
    unicode[6211]:=16#9633;
    unicode[6212]:=16#9634;
    unicode[6213]:=16#9635;
    unicode[6214]:=16#9636;
    unicode[6215]:=16#963b;
    unicode[6216]:=16#963c;
    unicode[6217]:=16#963d;
    unicode[6218]:=16#963f;
    unicode[6219]:=16#9640;
    unicode[6220]:=16#9642;
    unicode[6221]:=16#9644;
    unicode[6222]:=16#9645;
    unicode[6223]:=16#9646;
    unicode[6224]:=16#9647;
    unicode[6225]:=16#9648;
    unicode[6226]:=16#9649;
    unicode[6227]:=16#964b;
    unicode[6228]:=16#964c;
    unicode[6229]:=16#964d;
    unicode[6230]:=16#9650;
    unicode[6231]:=16#9654;
    unicode[6232]:=16#9655;
    unicode[6233]:=16#965b;
    unicode[6234]:=16#965f;
    unicode[6235]:=16#9661;
    unicode[6236]:=16#9662;
    unicode[6237]:=16#9664;
    unicode[6238]:=16#9667;
    unicode[6239]:=16#9668;
    unicode[6240]:=16#9669;
    unicode[6241]:=16#966a;
    unicode[6242]:=16#966c;
    unicode[6243]:=16#9672;
    unicode[6244]:=16#9674;
    unicode[6245]:=16#9675;
    unicode[6246]:=16#9676;
    unicode[6247]:=16#9677;
    unicode[6248]:=16#9685;
    unicode[6249]:=16#9686;
    unicode[6250]:=16#9688;
    unicode[6251]:=16#968b;
    unicode[6252]:=16#968d;
    unicode[6253]:=16#968f;
    unicode[6254]:=16#9690;
    unicode[6255]:=16#9694;
    unicode[6256]:=16#9697;
    unicode[6257]:=16#9698;
    unicode[6258]:=16#9699;
    unicode[6259]:=16#969c;
    unicode[6260]:=16#96a7;
    unicode[6261]:=16#96b0;
    unicode[6262]:=16#96b3;
    unicode[6263]:=16#96b6;
    unicode[6264]:=16#96b9;
    unicode[6265]:=16#96bc;
    unicode[6266]:=16#96bd;
    unicode[6267]:=16#96be;
    unicode[6268]:=16#96c0;
    unicode[6269]:=16#96c1;
    unicode[6270]:=16#96c4;
    unicode[6271]:=16#96c5;
    unicode[6272]:=16#96c6;
    unicode[6273]:=16#96c7;
    unicode[6274]:=16#96c9;
    unicode[6275]:=16#96cc;
    unicode[6276]:=16#96cd;
    unicode[6277]:=16#96ce;
    unicode[6278]:=16#96cf;
    unicode[6279]:=16#96d2;
    unicode[6280]:=16#96d5;
    unicode[6281]:=16#96e0;
    unicode[6282]:=16#96e8;
    unicode[6283]:=16#96e9;
    unicode[6284]:=16#96ea;
    unicode[6285]:=16#96ef;
    unicode[6286]:=16#96f3;
    unicode[6287]:=16#96f6;
    unicode[6288]:=16#96f7;
    unicode[6289]:=16#96f9;
    unicode[6290]:=16#96fe;
    unicode[6291]:=16#9700;
    unicode[6292]:=16#9701;
    unicode[6293]:=16#9704;
    unicode[6294]:=16#9706;
    unicode[6295]:=16#9707;
    unicode[6296]:=16#9708;
    unicode[6297]:=16#9709;
    unicode[6298]:=16#970d;
    unicode[6299]:=16#970e;
    unicode[6300]:=16#970f;
    unicode[6301]:=16#9713;
    unicode[6302]:=16#9716;
    unicode[6303]:=16#971c;
    unicode[6304]:=16#971e;
    unicode[6305]:=16#972a;
    unicode[6306]:=16#972d;
    unicode[6307]:=16#9730;
    unicode[6308]:=16#9732;
    unicode[6309]:=16#9738;
    unicode[6310]:=16#9739;
    unicode[6311]:=16#973e;
    unicode[6312]:=16#9752;
    unicode[6313]:=16#9753;
    unicode[6314]:=16#9756;
    unicode[6315]:=16#9759;
    unicode[6316]:=16#975b;
    unicode[6317]:=16#975e;
    unicode[6318]:=16#9760;
    unicode[6319]:=16#9761;
    unicode[6320]:=16#9762;
    unicode[6321]:=16#9765;
    unicode[6322]:=16#9769;
    unicode[6323]:=16#9773;
    unicode[6324]:=16#9774;
    unicode[6325]:=16#9776;
    unicode[6326]:=16#977c;
    unicode[6327]:=16#9785;
    unicode[6328]:=16#978b;
    unicode[6329]:=16#978d;
    unicode[6330]:=16#9791;
    unicode[6331]:=16#9792;
    unicode[6332]:=16#9794;
    unicode[6333]:=16#9798;
    unicode[6334]:=16#97a0;
    unicode[6335]:=16#97a3;
    unicode[6336]:=16#97ab;
    unicode[6337]:=16#97ad;
    unicode[6338]:=16#97af;
    unicode[6339]:=16#97b2;
    unicode[6340]:=16#97b4;
    unicode[6341]:=16#97e6;
    unicode[6342]:=16#97e7;
    unicode[6343]:=16#97e9;
    unicode[6344]:=16#97ea;
    unicode[6345]:=16#97eb;
    unicode[6346]:=16#97ec;
    unicode[6347]:=16#97ed;
    unicode[6348]:=16#97f3;
    unicode[6349]:=16#97f5;
    unicode[6350]:=16#97f6;
    unicode[6351]:=16#9875;
    unicode[6352]:=16#9876;
    unicode[6353]:=16#9877;
    unicode[6354]:=16#9878;
    unicode[6355]:=16#9879;
    unicode[6356]:=16#987a;
    unicode[6357]:=16#987b;
    unicode[6358]:=16#987c;
    unicode[6359]:=16#987d;
    unicode[6360]:=16#987e;
    unicode[6361]:=16#987f;
    unicode[6362]:=16#9880;
    unicode[6363]:=16#9881;
    unicode[6364]:=16#9882;
    unicode[6365]:=16#9883;
    unicode[6366]:=16#9884;
    unicode[6367]:=16#9885;
    unicode[6368]:=16#9886;
    unicode[6369]:=16#9887;
    unicode[6370]:=16#9888;
    unicode[6371]:=16#9889;
    unicode[6372]:=16#988a;
    unicode[6373]:=16#988c;
    unicode[6374]:=16#988d;
    unicode[6375]:=16#988f;
    unicode[6376]:=16#9890;
    unicode[6377]:=16#9891;
    unicode[6378]:=16#9893;
    unicode[6379]:=16#9894;
    unicode[6380]:=16#9896;
    unicode[6381]:=16#9897;
    unicode[6382]:=16#9898;
    unicode[6383]:=16#989a;
    unicode[6384]:=16#989b;
    unicode[6385]:=16#989c;
    unicode[6386]:=16#989d;
    unicode[6387]:=16#989e;
    unicode[6388]:=16#989f;
    unicode[6389]:=16#98a0;
    unicode[6390]:=16#98a1;
    unicode[6391]:=16#98a2;
    unicode[6392]:=16#98a4;
    unicode[6393]:=16#98a5;
    unicode[6394]:=16#98a6;
    unicode[6395]:=16#98a7;
    unicode[6396]:=16#98ce;
    unicode[6397]:=16#98d1;
    unicode[6398]:=16#98d2;
    unicode[6399]:=16#98d3;
    unicode[6400]:=16#98d5;
    unicode[6401]:=16#98d8;
    unicode[6402]:=16#98d9;
    unicode[6403]:=16#98da;
    unicode[6404]:=16#98de;
    unicode[6405]:=16#98df;
    unicode[6406]:=16#98e7;
    unicode[6407]:=16#98e8;
    unicode[6408]:=16#990d;
    unicode[6409]:=16#9910;
    unicode[6410]:=16#992e;
    unicode[6411]:=16#9954;
    unicode[6412]:=16#9955;
    unicode[6413]:=16#9963;
    unicode[6414]:=16#9965;
    unicode[6415]:=16#9967;
    unicode[6416]:=16#9968;
    unicode[6417]:=16#9969;
    unicode[6418]:=16#996a;
    unicode[6419]:=16#996b;
    unicode[6420]:=16#996c;
    unicode[6421]:=16#996d;
    unicode[6422]:=16#996e;
    unicode[6423]:=16#996f;
    unicode[6424]:=16#9970;
    unicode[6425]:=16#9971;
    unicode[6426]:=16#9972;
    unicode[6427]:=16#9974;
    unicode[6428]:=16#9975;
    unicode[6429]:=16#9976;
    unicode[6430]:=16#9977;
    unicode[6431]:=16#997a;
    unicode[6432]:=16#997c;
    unicode[6433]:=16#997d;
    unicode[6434]:=16#997f;
    unicode[6435]:=16#9980;
    unicode[6436]:=16#9981;
    unicode[6437]:=16#9984;
    unicode[6438]:=16#9985;
    unicode[6439]:=16#9986;
    unicode[6440]:=16#9987;
    unicode[6441]:=16#9988;
    unicode[6442]:=16#998a;
    unicode[6443]:=16#998b;
    unicode[6444]:=16#998d;
    unicode[6445]:=16#998f;
    unicode[6446]:=16#9990;
    unicode[6447]:=16#9991;
    unicode[6448]:=16#9992;
    unicode[6449]:=16#9993;
    unicode[6450]:=16#9994;
    unicode[6451]:=16#9995;
    unicode[6452]:=16#9996;
    unicode[6453]:=16#9997;
    unicode[6454]:=16#9998;
    unicode[6455]:=16#9999;
    unicode[6456]:=16#99a5;
    unicode[6457]:=16#99a8;
    unicode[6458]:=16#9a6c;
    unicode[6459]:=16#9a6d;
    unicode[6460]:=16#9a6e;
    unicode[6461]:=16#9a6f;
    unicode[6462]:=16#9a70;
    unicode[6463]:=16#9a71;
    unicode[6464]:=16#9a73;
    unicode[6465]:=16#9a74;
    unicode[6466]:=16#9a75;
    unicode[6467]:=16#9a76;
    unicode[6468]:=16#9a77;
    unicode[6469]:=16#9a78;
    unicode[6470]:=16#9a79;
    unicode[6471]:=16#9a7a;
    unicode[6472]:=16#9a7b;
    unicode[6473]:=16#9a7c;
    unicode[6474]:=16#9a7d;
    unicode[6475]:=16#9a7e;
    unicode[6476]:=16#9a7f;
    unicode[6477]:=16#9a80;
    unicode[6478]:=16#9a81;
    unicode[6479]:=16#9a82;
    unicode[6480]:=16#9a84;
    unicode[6481]:=16#9a85;
    unicode[6482]:=16#9a86;
    unicode[6483]:=16#9a87;
    unicode[6484]:=16#9a88;
    unicode[6485]:=16#9a8a;
    unicode[6486]:=16#9a8b;
    unicode[6487]:=16#9a8c;
    unicode[6488]:=16#9a8f;
    unicode[6489]:=16#9a90;
    unicode[6490]:=16#9a91;
    unicode[6491]:=16#9a92;
    unicode[6492]:=16#9a93;
    unicode[6493]:=16#9a96;
    unicode[6494]:=16#9a97;
    unicode[6495]:=16#9a98;
    unicode[6496]:=16#9a9a;
    unicode[6497]:=16#9a9b;
    unicode[6498]:=16#9a9c;
    unicode[6499]:=16#9a9d;
    unicode[6500]:=16#9a9e;
    unicode[6501]:=16#9a9f;
    unicode[6502]:=16#9aa0;
    unicode[6503]:=16#9aa1;
    unicode[6504]:=16#9aa2;
    unicode[6505]:=16#9aa3;
    unicode[6506]:=16#9aa4;
    unicode[6507]:=16#9aa5;
    unicode[6508]:=16#9aa7;
    unicode[6509]:=16#9aa8;
    unicode[6510]:=16#9ab0;
    unicode[6511]:=16#9ab1;
    unicode[6512]:=16#9ab6;
    unicode[6513]:=16#9ab7;
    unicode[6514]:=16#9ab8;
    unicode[6515]:=16#9aba;
    unicode[6516]:=16#9abc;
    unicode[6517]:=16#9ac0;
    unicode[6518]:=16#9ac1;
    unicode[6519]:=16#9ac2;
    unicode[6520]:=16#9ac5;
    unicode[6521]:=16#9acb;
    unicode[6522]:=16#9acc;
    unicode[6523]:=16#9ad1;
    unicode[6524]:=16#9ad3;
    unicode[6525]:=16#9ad8;
    unicode[6526]:=16#9adf;
    unicode[6527]:=16#9ae1;
    unicode[6528]:=16#9ae6;
    unicode[6529]:=16#9aeb;
    unicode[6530]:=16#9aed;
    unicode[6531]:=16#9aef;
    unicode[6532]:=16#9af9;
    unicode[6533]:=16#9afb;
    unicode[6534]:=16#9b03;
    unicode[6535]:=16#9b08;
    unicode[6536]:=16#9b0f;
    unicode[6537]:=16#9b13;
    unicode[6538]:=16#9b1f;
    unicode[6539]:=16#9b23;
    unicode[6540]:=16#9b2f;
    unicode[6541]:=16#9b32;
    unicode[6542]:=16#9b3b;
    unicode[6543]:=16#9b3c;
    unicode[6544]:=16#9b41;
    unicode[6545]:=16#9b42;
    unicode[6546]:=16#9b43;
    unicode[6547]:=16#9b44;
    unicode[6548]:=16#9b45;
    unicode[6549]:=16#9b47;
    unicode[6550]:=16#9b48;
    unicode[6551]:=16#9b49;
    unicode[6552]:=16#9b4d;
    unicode[6553]:=16#9b4f;
    unicode[6554]:=16#9b51;
    unicode[6555]:=16#9b54;
    unicode[6556]:=16#9c7c;
    unicode[6557]:=16#9c7f;
    unicode[6558]:=16#9c81;
    unicode[6559]:=16#9c82;
    unicode[6560]:=16#9c85;
    unicode[6561]:=16#9c86;
    unicode[6562]:=16#9c87;
    unicode[6563]:=16#9c88;
    unicode[6564]:=16#9c8b;
    unicode[6565]:=16#9c8d;
    unicode[6566]:=16#9c8e;
    unicode[6567]:=16#9c90;
    unicode[6568]:=16#9c91;
    unicode[6569]:=16#9c92;
    unicode[6570]:=16#9c94;
    unicode[6571]:=16#9c95;
    unicode[6572]:=16#9c9a;
    unicode[6573]:=16#9c9b;
    unicode[6574]:=16#9c9c;
    unicode[6575]:=16#9c9e;
    unicode[6576]:=16#9c9f;
    unicode[6577]:=16#9ca0;
    unicode[6578]:=16#9ca1;
    unicode[6579]:=16#9ca2;
    unicode[6580]:=16#9ca3;
    unicode[6581]:=16#9ca4;
    unicode[6582]:=16#9ca5;
    unicode[6583]:=16#9ca6;
    unicode[6584]:=16#9ca7;
    unicode[6585]:=16#9ca8;
    unicode[6586]:=16#9ca9;
    unicode[6587]:=16#9cab;
    unicode[6588]:=16#9cad;
    unicode[6589]:=16#9cae;
    unicode[6590]:=16#9cb0;
    unicode[6591]:=16#9cb1;
    unicode[6592]:=16#9cb2;
    unicode[6593]:=16#9cb3;
    unicode[6594]:=16#9cb4;
    unicode[6595]:=16#9cb5;
    unicode[6596]:=16#9cb6;
    unicode[6597]:=16#9cb7;
    unicode[6598]:=16#9cb8;
    unicode[6599]:=16#9cba;
    unicode[6600]:=16#9cbb;
    unicode[6601]:=16#9cbc;
    unicode[6602]:=16#9cbd;
    unicode[6603]:=16#9cc3;
    unicode[6604]:=16#9cc4;
    unicode[6605]:=16#9cc5;
    unicode[6606]:=16#9cc6;
    unicode[6607]:=16#9cc7;
    unicode[6608]:=16#9cca;
    unicode[6609]:=16#9ccb;
    unicode[6610]:=16#9ccc;
    unicode[6611]:=16#9ccd;
    unicode[6612]:=16#9cce;
    unicode[6613]:=16#9ccf;
    unicode[6614]:=16#9cd0;
    unicode[6615]:=16#9cd3;
    unicode[6616]:=16#9cd4;
    unicode[6617]:=16#9cd5;
    unicode[6618]:=16#9cd6;
    unicode[6619]:=16#9cd7;
    unicode[6620]:=16#9cd8;
    unicode[6621]:=16#9cd9;
    unicode[6622]:=16#9cdc;
    unicode[6623]:=16#9cdd;
    unicode[6624]:=16#9cde;
    unicode[6625]:=16#9cdf;
    unicode[6626]:=16#9ce2;
    unicode[6627]:=16#9e1f;
    unicode[6628]:=16#9e20;
    unicode[6629]:=16#9e21;
    unicode[6630]:=16#9e22;
    unicode[6631]:=16#9e23;
    unicode[6632]:=16#9e25;
    unicode[6633]:=16#9e26;
    unicode[6634]:=16#9e28;
    unicode[6635]:=16#9e29;
    unicode[6636]:=16#9e2a;
    unicode[6637]:=16#9e2b;
    unicode[6638]:=16#9e2c;
    unicode[6639]:=16#9e2d;
    unicode[6640]:=16#9e2f;
    unicode[6641]:=16#9e31;
    unicode[6642]:=16#9e32;
    unicode[6643]:=16#9e33;
    unicode[6644]:=16#9e35;
    unicode[6645]:=16#9e36;
    unicode[6646]:=16#9e37;
    unicode[6647]:=16#9e38;
    unicode[6648]:=16#9e39;
    unicode[6649]:=16#9e3a;
    unicode[6650]:=16#9e3d;
    unicode[6651]:=16#9e3e;
    unicode[6652]:=16#9e3f;
    unicode[6653]:=16#9e41;
    unicode[6654]:=16#9e42;
    unicode[6655]:=16#9e43;
    unicode[6656]:=16#9e44;
    unicode[6657]:=16#9e45;
    unicode[6658]:=16#9e46;
    unicode[6659]:=16#9e47;
    unicode[6660]:=16#9e48;
    unicode[6661]:=16#9e49;
    unicode[6662]:=16#9e4a;
    unicode[6663]:=16#9e4b;
    unicode[6664]:=16#9e4c;
    unicode[6665]:=16#9e4e;
    unicode[6666]:=16#9e4f;
    unicode[6667]:=16#9e51;
    unicode[6668]:=16#9e55;
    unicode[6669]:=16#9e57;
    unicode[6670]:=16#9e58;
    unicode[6671]:=16#9e5a;
    unicode[6672]:=16#9e5b;
    unicode[6673]:=16#9e5c;
    unicode[6674]:=16#9e5e;
    unicode[6675]:=16#9e63;
    unicode[6676]:=16#9e64;
    unicode[6677]:=16#9e66;
    unicode[6678]:=16#9e67;
    unicode[6679]:=16#9e68;
    unicode[6680]:=16#9e69;
    unicode[6681]:=16#9e6a;
    unicode[6682]:=16#9e6b;
    unicode[6683]:=16#9e6c;
    unicode[6684]:=16#9e6d;
    unicode[6685]:=16#9e70;
    unicode[6686]:=16#9e71;
    unicode[6687]:=16#9e73;
    unicode[6688]:=16#9e7e;
    unicode[6689]:=16#9e7f;
    unicode[6690]:=16#9e82;
    unicode[6691]:=16#9e87;
    unicode[6692]:=16#9e88;
    unicode[6693]:=16#9e8b;
    unicode[6694]:=16#9e92;
    unicode[6695]:=16#9e93;
    unicode[6696]:=16#9e9d;
    unicode[6697]:=16#9e9f;
    unicode[6698]:=16#9ea6;
    unicode[6699]:=16#9eb4;
    unicode[6700]:=16#9eb8;
    unicode[6701]:=16#9ebb;
    unicode[6702]:=16#9ebd;
    unicode[6703]:=16#9ebe;
    unicode[6704]:=16#9ec4;
    unicode[6705]:=16#9ec9;
    unicode[6706]:=16#9ecd;
    unicode[6707]:=16#9ece;
    unicode[6708]:=16#9ecf;
    unicode[6709]:=16#9ed1;
    unicode[6710]:=16#9ed4;
    unicode[6711]:=16#9ed8;
    unicode[6712]:=16#9edb;
    unicode[6713]:=16#9edc;
    unicode[6714]:=16#9edd;
    unicode[6715]:=16#9edf;
    unicode[6716]:=16#9ee0;
    unicode[6717]:=16#9ee2;
    unicode[6718]:=16#9ee5;
    unicode[6719]:=16#9ee7;
    unicode[6720]:=16#9ee9;
    unicode[6721]:=16#9eea;
    unicode[6722]:=16#9eef;
    unicode[6723]:=16#9ef9;
    unicode[6724]:=16#9efb;
    unicode[6725]:=16#9efc;
    unicode[6726]:=16#9efe;
    unicode[6727]:=16#9f0b;
    unicode[6728]:=16#9f0d;
    unicode[6729]:=16#9f0e;
    unicode[6730]:=16#9f10;
    unicode[6731]:=16#9f13;
    unicode[6732]:=16#9f17;
    unicode[6733]:=16#9f19;
    unicode[6734]:=16#9f20;
    unicode[6735]:=16#9f22;
    unicode[6736]:=16#9f2c;
    unicode[6737]:=16#9f2f;
    unicode[6738]:=16#9f37;
    unicode[6739]:=16#9f39;
    unicode[6740]:=16#9f3b;
    unicode[6741]:=16#9f3d;
    unicode[6742]:=16#9f3e;
    unicode[6743]:=16#9f44;
    unicode[6744]:=16#9f50;
    unicode[6745]:=16#9f51;
    unicode[6746]:=16#9f7f;
    unicode[6747]:=16#9f80;
    unicode[6748]:=16#9f83;
    unicode[6749]:=16#9f84;
    unicode[6750]:=16#9f85;
    unicode[6751]:=16#9f86;
    unicode[6752]:=16#9f87;
    unicode[6753]:=16#9f88;
    unicode[6754]:=16#9f89;
    unicode[6755]:=16#9f8a;
    unicode[6756]:=16#9f8b;
    unicode[6757]:=16#9f8c;
    unicode[6758]:=16#9f99;
    unicode[6759]:=16#9f9a;
    unicode[6760]:=16#9f9b;
    unicode[6761]:=16#9f9f;
    unicode[6762]:=16#9fa0;
    unicode[6763]:=16#e810;
    unicode[6764]:=16#e811;
    unicode[6765]:=16#e812;
    unicode[6766]:=16#e813;
    unicode[6767]:=16#e814;
    unicode[6768]:=16#ff01;
    unicode[6769]:=16#ff08;
    unicode[6770]:=16#ff09;
    unicode[6771]:=16#ff0c;
    unicode[6772]:=16#ff1a;
    unicode[6773]:=16#ff1b;
    unicode[6774]:=16#ff1f;
    unicode[6775]:=16#ffe5;           //unicode码 6000-6999
END_IF;
(* Rung 11 *)
IF P_On THEN
    GB2312[0]:= 16#d2bb;
    GB2312[1]:= 16#b6a1;
    GB2312[2]:= 16#c6df;
    GB2312[3]:= 16#cdf2;
    GB2312[4]:= 16#d5c9;
    GB2312[5]:= 16#c8fd;
    GB2312[6]:= 16#c9cf;
    GB2312[7]:= 16#cfc2;
    GB2312[8]:= 16#d8a2;
    GB2312[9]:= 16#b2bb;
    GB2312[10]:= 16#d3eb;
    GB2312[11]:= 16#d8a4;
    GB2312[12]:= 16#b3f3;
    GB2312[13]:= 16#d7a8;
    GB2312[14]:= 16#c7d2;
    GB2312[15]:= 16#d8a7;
    GB2312[16]:= 16#cac0;
    GB2312[17]:= 16#c7f0;
    GB2312[18]:= 16#b1fb;
    GB2312[19]:= 16#d2b5;
    GB2312[20]:= 16#b4d4;
    GB2312[21]:= 16#b6ab;
    GB2312[22]:= 16#cbbf;
    GB2312[23]:= 16#d8a9;
    GB2312[24]:= 16#b6aa;
    GB2312[25]:= 16#c1bd;
    GB2312[26]:= 16#d1cf;
    GB2312[27]:= 16#c9a5;
    GB2312[28]:= 16#d8ad;
    GB2312[29]:= 16#b8f6;
    GB2312[30]:= 16#d1be;
    GB2312[31]:= 16#e3dc;
    GB2312[32]:= 16#d6d0;
    GB2312[33]:= 16#b7e1;
    GB2312[34]:= 16#b4ae;
    GB2312[35]:= 16#c1d9;
    GB2312[36]:= 16#d8bc;
    GB2312[37]:= 16#cde8;
    GB2312[38]:= 16#b5a4;
    GB2312[39]:= 16#ceaa;
    GB2312[40]:= 16#d6f7;
    GB2312[41]:= 16#c0f6;
    GB2312[42]:= 16#bed9;
    GB2312[43]:= 16#d8af;
    GB2312[44]:= 16#c4cb;
    GB2312[45]:= 16#bec3;
    GB2312[46]:= 16#d8b1;
    GB2312[47]:= 16#c3b4;
    GB2312[48]:= 16#d2e5;
    GB2312[49]:= 16#d6ae;
    GB2312[50]:= 16#ceda;
    GB2312[51]:= 16#d5a7;
    GB2312[52]:= 16#baf5;
    GB2312[53]:= 16#b7a6;
    GB2312[54]:= 16#c0d6;
    GB2312[55]:= 16#c6b9;
    GB2312[56]:= 16#c5d2;
    GB2312[57]:= 16#c7c7;
    GB2312[58]:= 16#b9d4;
    GB2312[59]:= 16#b3cb;
    GB2312[60]:= 16#d2d2;
    GB2312[61]:= 16#d8bf;
    GB2312[62]:= 16#bec5;
    GB2312[63]:= 16#c6f2;
    GB2312[64]:= 16#d2b2;
    GB2312[65]:= 16#cfb0;
    GB2312[66]:= 16#cfe7;
    GB2312[67]:= 16#cae9;
    GB2312[68]:= 16#d8c0;
    GB2312[69]:= 16#c2f2;
    GB2312[70]:= 16#c2d2;
    GB2312[71]:= 16#c8e9;
    GB2312[72]:= 16#c7ac;
    GB2312[73]:= 16#c1cb;
    GB2312[74]:= 16#d3e8;
    GB2312[75]:= 16#d5f9;
    GB2312[76]:= 16#cac2;
    GB2312[77]:= 16#b6fe;
    GB2312[78]:= 16#d8a1;
    GB2312[79]:= 16#d3da;
    GB2312[80]:= 16#bff7;
    GB2312[81]:= 16#d4c6;
    GB2312[82]:= 16#bba5;
    GB2312[83]:= 16#d8c1;
    GB2312[84]:= 16#cee5;
    GB2312[85]:= 16#beae;
    GB2312[86]:= 16#d8a8;
    GB2312[87]:= 16#d1c7;
    GB2312[88]:= 16#d0a9;
    GB2312[89]:= 16#d8bd;
    GB2312[90]:= 16#d9ef;
    GB2312[91]:= 16#cdf6;
    GB2312[92]:= 16#bfba;
    GB2312[93]:= 16#bdbb;
    GB2312[94]:= 16#baa5;
    GB2312[95]:= 16#d2e0;
    GB2312[96]:= 16#b2fa;
    GB2312[97]:= 16#bae0;
    GB2312[98]:= 16#c4b6;
    GB2312[99]:= 16#cfed;
    GB2312[100]:= 16#bea9;
    GB2312[101]:= 16#cda4;
    GB2312[102]:= 16#c1c1;
    GB2312[103]:= 16#c7d7;
    GB2312[104]:= 16#d9f1;
    GB2312[105]:= 16#d9f4;
    GB2312[106]:= 16#c8cb;
    GB2312[107]:= 16#d8e9;
    GB2312[108]:= 16#d2da;
    GB2312[109]:= 16#cab2;
    GB2312[110]:= 16#c8ca;
    GB2312[111]:= 16#d8ec;
    GB2312[112]:= 16#d8ea;
    GB2312[113]:= 16#d8c6;
    GB2312[114]:= 16#bdf6;
    GB2312[115]:= 16#c6cd;
    GB2312[116]:= 16#b3f0;
    GB2312[117]:= 16#d8eb;
    GB2312[118]:= 16#bdf1;
    GB2312[119]:= 16#bde9;
    GB2312[120]:= 16#c8d4;
    GB2312[121]:= 16#b4d3;
    GB2312[122]:= 16#c2d8;
    GB2312[123]:= 16#b2d6;
    GB2312[124]:= 16#d7d0;
    GB2312[125]:= 16#cacb;
    GB2312[126]:= 16#cbfb;
    GB2312[127]:= 16#d5cc;
    GB2312[128]:= 16#b8b6;
    GB2312[129]:= 16#cfc9;
    GB2312[130]:= 16#d9da;
    GB2312[131]:= 16#d8f0;
    GB2312[132]:= 16#c7aa;
    GB2312[133]:= 16#d8ee;
    GB2312[134]:= 16#b4fa;
    GB2312[135]:= 16#c1ee;
    GB2312[136]:= 16#d2d4;
    GB2312[137]:= 16#d8ed;
    GB2312[138]:= 16#d2c7;
    GB2312[139]:= 16#d8ef;
    GB2312[140]:= 16#c3c7;
    GB2312[141]:= 16#d1f6;
    GB2312[142]:= 16#d6d9;
    GB2312[143]:= 16#d8f2;
    GB2312[144]:= 16#d8f5;
    GB2312[145]:= 16#bcfe;
    GB2312[146]:= 16#bcdb;
    GB2312[147]:= 16#c8ce;
    GB2312[148]:= 16#b7dd;
    GB2312[149]:= 16#b7c2;
    GB2312[150]:= 16#c6f3;
    GB2312[151]:= 16#d8f8;
    GB2312[152]:= 16#d2c1;
    GB2312[153]:= 16#cee9;
    GB2312[154]:= 16#bcbf;
    GB2312[155]:= 16#b7fc;
    GB2312[156]:= 16#b7a5;
    GB2312[157]:= 16#d0dd;
    GB2312[158]:= 16#d6da;
    GB2312[159]:= 16#d3c5;
    GB2312[160]:= 16#bbef;
    GB2312[161]:= 16#bbe1;
    GB2312[162]:= 16#d8f1;
    GB2312[163]:= 16#c9a1;
    GB2312[164]:= 16#ceb0;
    GB2312[165]:= 16#b4ab;
    GB2312[166]:= 16#d8f3;
    GB2312[167]:= 16#c9cb;
    GB2312[168]:= 16#d8f6;
    GB2312[169]:= 16#c2d7;
    GB2312[170]:= 16#d8f7;
    GB2312[171]:= 16#ceb1;
    GB2312[172]:= 16#d8f9;
    GB2312[173]:= 16#b2ae;
    GB2312[174]:= 16#b9c0;
    GB2312[175]:= 16#d9a3;
    GB2312[176]:= 16#b0e9;
    GB2312[177]:= 16#c1e6;
    GB2312[178]:= 16#c9ec;
    GB2312[179]:= 16#cbc5;
    GB2312[180]:= 16#cbc6;
    GB2312[181]:= 16#d9a4;
    GB2312[182]:= 16#b5e8;
    GB2312[183]:= 16#b5ab;
    GB2312[184]:= 16#cebb;
    GB2312[185]:= 16#b5cd;
    GB2312[186]:= 16#d7a1;
    GB2312[187]:= 16#d7f4;
    GB2312[188]:= 16#d3d3;
    GB2312[189]:= 16#cce5;
    GB2312[190]:= 16#bace;
    GB2312[191]:= 16#d9a2;
    GB2312[192]:= 16#d9dc;
    GB2312[193]:= 16#d3e0;
    GB2312[194]:= 16#d8fd;
    GB2312[195]:= 16#b7f0;
    GB2312[196]:= 16#d7f7;
    GB2312[197]:= 16#d8fe;
    GB2312[198]:= 16#d8fa;
    GB2312[199]:= 16#d9a1;
    GB2312[200]:= 16#c4e3;
    GB2312[201]:= 16#d3b6;
    GB2312[202]:= 16#d8f4;
    GB2312[203]:= 16#d9dd;
    GB2312[204]:= 16#d8fb;
    GB2312[205]:= 16#c5e5;
    GB2312[206]:= 16#c0d0;
    GB2312[207]:= 16#d1f0;
    GB2312[208]:= 16#b0db;
    GB2312[209]:= 16#bcd1;
    GB2312[210]:= 16#d9a6;
    GB2312[211]:= 16#d9a5;
    GB2312[212]:= 16#d9ac;
    GB2312[213]:= 16#d9ae;
    GB2312[214]:= 16#d9ab;
    GB2312[215]:= 16#cab9;
    GB2312[216]:= 16#d9a9;
    GB2312[217]:= 16#d6b6;
    GB2312[218]:= 16#b3de;
    GB2312[219]:= 16#d9a8;
    GB2312[220]:= 16#c0fd;
    GB2312[221]:= 16#cacc;
    GB2312[222]:= 16#d9aa;
    GB2312[223]:= 16#d9a7;
    GB2312[224]:= 16#d9b0;
    GB2312[225]:= 16#b6b1;
    GB2312[226]:= 16#b9a9;
    GB2312[227]:= 16#d2c0;
    GB2312[228]:= 16#cfc0;
    GB2312[229]:= 16#c2c2;
    GB2312[230]:= 16#bdc4;
    GB2312[231]:= 16#d5ec;
    GB2312[232]:= 16#b2e0;
    GB2312[233]:= 16#c7c8;
    GB2312[234]:= 16#bfeb;
    GB2312[235]:= 16#d9ad;
    GB2312[236]:= 16#d9af;
    GB2312[237]:= 16#ceea;
    GB2312[238]:= 16#baee;
    GB2312[239]:= 16#c7d6;
    GB2312[240]:= 16#b1e3;
    GB2312[241]:= 16#b4d9;
    GB2312[242]:= 16#b6ed;
    GB2312[243]:= 16#d9b4;
    GB2312[244]:= 16#bfa1;
    GB2312[245]:= 16#d9de;
    GB2312[246]:= 16#c7ce;
    GB2312[247]:= 16#c0fe;
    GB2312[248]:= 16#d9b8;
    GB2312[249]:= 16#cbd7;
    GB2312[250]:= 16#b7fd;
    GB2312[251]:= 16#d9b5;
    GB2312[252]:= 16#d9b7;
    GB2312[253]:= 16#b1a3;
    GB2312[254]:= 16#d3e1;
    GB2312[255]:= 16#d9b9;
    GB2312[256]:= 16#d0c5;
    GB2312[257]:= 16#d9b6;
    GB2312[258]:= 16#d9b1;
    GB2312[259]:= 16#d9b2;
    GB2312[260]:= 16#c1a9;
    GB2312[261]:= 16#d9b3;
    GB2312[262]:= 16#bcf3;
    GB2312[263]:= 16#d0de;
    GB2312[264]:= 16#b8a9;
    GB2312[265]:= 16#bee3;
    GB2312[266]:= 16#d9bd;
    GB2312[267]:= 16#d9ba;
    GB2312[268]:= 16#b0b3;
    GB2312[269]:= 16#d9c2;
    GB2312[270]:= 16#d9c4;
    GB2312[271]:= 16#b1b6;
    GB2312[272]:= 16#d9bf;
    GB2312[273]:= 16#b5b9;
    GB2312[274]:= 16#bef3;
    GB2312[275]:= 16#ccc8;
    GB2312[276]:= 16#baf2;
    GB2312[277]:= 16#d2d0;
    GB2312[278]:= 16#d9c3;
    GB2312[279]:= 16#bde8;
    GB2312[280]:= 16#b3ab;
    GB2312[281]:= 16#d9c5;
    GB2312[282]:= 16#beeb;
    GB2312[283]:= 16#d9c6;
    GB2312[284]:= 16#d9bb;
    GB2312[285]:= 16#c4df;
    GB2312[286]:= 16#d9be;
    GB2312[287]:= 16#d9c1;
    GB2312[288]:= 16#d9c0;
    GB2312[289]:= 16#d5ae;
    GB2312[290]:= 16#d6b5;
    GB2312[291]:= 16#c7e3;
    GB2312[292]:= 16#d9c8;
    GB2312[293]:= 16#bcd9;
    GB2312[294]:= 16#d9ca;
    GB2312[295]:= 16#d9bc;
    GB2312[296]:= 16#d9cb;
    GB2312[297]:= 16#c6ab;
    GB2312[298]:= 16#d9c9;
    GB2312[299]:= 16#d7f6;
    GB2312[300]:= 16#cda3;
    GB2312[301]:= 16#bda1;
    GB2312[302]:= 16#d9cc;
    GB2312[303]:= 16#c5bc;
    GB2312[304]:= 16#cdb5;
    GB2312[305]:= 16#d9cd;
    GB2312[306]:= 16#d9c7;
    GB2312[307]:= 16#b3a5;
    GB2312[308]:= 16#bffe;
    GB2312[309]:= 16#b8b5;
    GB2312[310]:= 16#c0fc;
    GB2312[311]:= 16#b0f8;
    GB2312[312]:= 16#b4f6;
    GB2312[313]:= 16#d9ce;
    GB2312[314]:= 16#d9cf;
    GB2312[315]:= 16#b4a2;
    GB2312[316]:= 16#d9d0;
    GB2312[317]:= 16#b4df;
    GB2312[318]:= 16#b0c1;
    GB2312[319]:= 16#d9d1;
    GB2312[320]:= 16#c9b5;
    GB2312[321]:= 16#cff1;
    GB2312[322]:= 16#d9d2;
    GB2312[323]:= 16#c1c5;
    GB2312[324]:= 16#d9d6;
    GB2312[325]:= 16#c9ae;
    GB2312[326]:= 16#d9d5;
    GB2312[327]:= 16#d9d4;
    GB2312[328]:= 16#d9d7;
    GB2312[329]:= 16#cbdb;
    GB2312[330]:= 16#bda9;
    GB2312[331]:= 16#c6a7;
    GB2312[332]:= 16#d9d3;
    GB2312[333]:= 16#d9d8;
    GB2312[334]:= 16#d9d9;
    GB2312[335]:= 16#c8e5;
    GB2312[336]:= 16#c0dc;
    GB2312[337]:= 16#b6f9;
    GB2312[338]:= 16#d8a3;
    GB2312[339]:= 16#d4ca;
    GB2312[340]:= 16#d4aa;
    GB2312[341]:= 16#d0d6;
    GB2312[342]:= 16#b3e4;
    GB2312[343]:= 16#d5d7;
    GB2312[344]:= 16#cfc8;
    GB2312[345]:= 16#b9e2;
    GB2312[346]:= 16#bfcb;
    GB2312[347]:= 16#c3e2;
    GB2312[348]:= 16#b6d2;
    GB2312[349]:= 16#cdc3;
    GB2312[350]:= 16#d9ee;
    GB2312[351]:= 16#d9f0;
    GB2312[352]:= 16#b5b3;
    GB2312[353]:= 16#b6b5;
    GB2312[354]:= 16#bea4;
    GB2312[355]:= 16#c8eb;
    GB2312[356]:= 16#c8ab;
    GB2312[357]:= 16#b0cb;
    GB2312[358]:= 16#b9ab;
    GB2312[359]:= 16#c1f9;
    GB2312[360]:= 16#d9e2;
    GB2312[361]:= 16#c0bc;
    GB2312[362]:= 16#b9b2;
    GB2312[363]:= 16#b9d8;
    GB2312[364]:= 16#d0cb;
    GB2312[365]:= 16#b1f8;
    GB2312[366]:= 16#c6e4;
    GB2312[367]:= 16#bedf;
    GB2312[368]:= 16#b5e4;
    GB2312[369]:= 16#d7c8;
    GB2312[370]:= 16#d1f8;
    GB2312[371]:= 16#bce6;
    GB2312[372]:= 16#cade;
    GB2312[373]:= 16#bcbd;
    GB2312[374]:= 16#d9e6;
    GB2312[375]:= 16#d8e7;
    GB2312[376]:= 16#c4da;
    GB2312[377]:= 16#b8d4;
    GB2312[378]:= 16#c8bd;
    GB2312[379]:= 16#b2e1;
    GB2312[380]:= 16#d4d9;
    GB2312[381]:= 16#c3b0;
    GB2312[382]:= 16#c3e1;
    GB2312[383]:= 16#daa2;
    GB2312[384]:= 16#c8df;
    GB2312[385]:= 16#d0b4;
    GB2312[386]:= 16#befc;
    GB2312[387]:= 16#c5a9;
    GB2312[388]:= 16#b9da;
    GB2312[389]:= 16#daa3;
    GB2312[390]:= 16#d4a9;
    GB2312[391]:= 16#daa4;
    GB2312[392]:= 16#d9fb;
    GB2312[393]:= 16#b6ac;
    GB2312[394]:= 16#b7eb;
    GB2312[395]:= 16#b1f9;
    GB2312[396]:= 16#d9fc;
    GB2312[397]:= 16#b3e5;
